               "gtyp_VGR".vertical_Axis.di_Target_Position := "gtyp_VGR".di_Pos_NFC_vertical - "gtyp_VGR".di_Offset_Pos_DSI_NFC_vertical;
               "gtyp_VGR".vertical_Axis.x_Start_Positioning := TRUE;
               //"gtyp_VGR".vertical_Axis.i_PWM := 800;

               IF ("gtyp_VGR".vertical_Axis.di_Actual_Position <= ("gtyp_VGR".di_Pos_NFC_vertical - "gtyp_VGR".di_Offset_Pos_DSI_NFC_vertical + "gtyp_VGR".vertical_Axis.Config.di_Pos_Window))
                   AND ("gtyp_VGR".vertical_Axis.di_Actual_Position >= ("gtyp_VGR".di_Pos_NFC_vertical - "gtyp_VGR".di_Offset_Pos_DSI_NFC_vertical - "gtyp_VGR".vertical_Axis.Config.di_Pos_Window))
                   AND "gtyp_VGR".vertical_Axis.x_Position_Reached THEN
                   "gtyp_VGR".vertical_Axis.x_Start_Positioning := FALSE;
                   #li_StepCase := 660;
               END_IF;

           660: // wait sequence
               #lx_Start_TON_Wait := TRUE;
               #lt_TON_Wait := T#500ms;

               IF #lfb_TON_Wait.Q THEN
                   #lx_Start_TON_Wait := FALSE;
                   #li_StepCase := 670;
               END_IF;

           670: // Position horizontal/rotate NFC

               "gtyp_VGR".horizontal_Axis.di_Target_Position := "gtyp_VGR".di_Pos_NFC_horizontal;
               "gtyp_VGR".horizontal_Axis.x_Start_Positioning := TRUE;
               "gtyp_VGR".rotate_Axis.di_Target_Position := "gtyp_VGR".di_Pos_NFC_rotate;
               "gtyp_VGR".rotate_Axis.x_Start_Positioning := TRUE;

               IF ("gtyp_VGR".horizontal_Axis.di_Actual_Position <= ("gtyp_VGR".di_Pos_NFC_horizontal + "gtyp_VGR".horizontal_Axis.Config.di_Pos_Window))
                   AND ("gtyp_VGR".horizontal_Axis.di_Actual_Position >= ("gtyp_VGR".di_Pos_NFC_horizontal - "gtyp_VGR".horizontal_Axis.Config.di_Pos_Window))
                   AND "gtyp_VGR".horizontal_Axis.x_Position_Reached THEN
                   "gtyp_VGR".horizontal_Axis.x_Start_Positioning := FALSE;
               END_IF;

               IF ("gtyp_VGR".rotate_Axis.di_Actual_Position <= ("gtyp_VGR".di_Pos_NFC_rotate + "gtyp_VGR".rotate_Axis.Config.di_Pos_Window))
                   AND ("gtyp_VGR".rotate_Axis.di_Actual_Position >= ("gtyp_VGR".di_Pos_NFC_rotate - "gtyp_VGR".rotate_Axis.Config.di_Pos_Window))
                   AND "gtyp_VGR".rotate_Axis.x_Position_Reached THEN
                   "gtyp_VGR".rotate_Axis.x_Start_Positioning := FALSE;
               END_IF;

               IF ("gtyp_VGR".horizontal_Axis.di_Actual_Position <= ("gtyp_VGR".di_Pos_NFC_horizontal + "gtyp_VGR".horizontal_Axis.Config.di_Pos_Window))
                   AND ("gtyp_VGR".horizontal_Axis.di_Actual_Position >= ("gtyp_VGR".di_Pos_NFC_horizontal - "gtyp_VGR".horizontal_Axis.Config.di_Pos_Window))
                   AND "gtyp_VGR".horizontal_Axis.x_Position_Reached
                   AND ("gtyp_VGR".rotate_Axis.di_Actual_Position <= ("gtyp_VGR".di_Pos_NFC_rotate + "gtyp_VGR".rotate_Axis.Config.di_Pos_Window))
                   AND ("gtyp_VGR".rotate_Axis.di_Actual_Position >= ("gtyp_VGR".di_Pos_NFC_rotate - "gtyp_VGR".rotate_Axis.Config.di_Pos_Window))
                   AND "gtyp_VGR".rotate_Axis.x_Position_Reached THEN
                   "gtyp_VGR".horizontal_Axis.x_Start_Positioning := FALSE;
                   "gtyp_VGR".rotate_Axis.x_Start_Positioning := FALSE;
                   #li_StepCase := 680;
               END_IF;

           680: // wait sequence
               #lx_Start_TON_Wait := TRUE;
               #lt_TON_Wait := T#500ms;

               IF #lfb_TON_Wait.Q THEN
                   #lx_Start_TON_Wait := FALSE;
                   #li_StepCase := 690;
               END_IF;

           690: // Position vertical NFC

               "gtyp_VGR".vertical_Axis.di_Target_Position := "gtyp_VGR".di_Pos_NFC_vertical;
               "gtyp_VGR".vertical_Axis.x_Start_Positioning := TRUE;
               //"gtyp_VGR".vertical_Axis.i_PWM := 500;

               IF ("gtyp_VGR".vertical_Axis.di_Actual_Position <= ("gtyp_VGR".di_Pos_NFC_vertical + "gtyp_VGR".vertical_Axis.Config.di_Pos_Window))
                   AND ("gtyp_VGR".vertical_Axis.di_Actual_Position >= ("gtyp_VGR".di_Pos_NFC_vertical - "gtyp_VGR".vertical_Axis.Config.di_Pos_Window))
                   AND "gtyp_VGR".vertical_Axis.x_Position_Reached THEN
                   "gtyp_VGR".vertical_Axis.x_Start_Positioning := FALSE;
                   //"gtyp_VGR".vertical_Axis.i_PWM := 800;
                   #li_StepCase := 700;
               END_IF;

           700: // Start delete/write/read NFC 
               "gtyp_VGR".x_NFC_Start_First := TRUE;

               IF "gtyp_VGR".x_NFC_Completed THEN
                   "gtyp_VGR".x_NFC_Start_First := FALSE;
                   #li_StepCase := 710;
               END_IF;

           710: // Position vertical pre NFC

               "gtyp_VGR".vertical_Axis.di_Target_Position := "gtyp_VGR".di_Pos_NFC_vertical - "gtyp_VGR".di_Offset_Pos_DSI_NFC_vertical;
               "gtyp_VGR".vertical_Axis.x_Start_Positioning := TRUE;
               //"gtyp_VGR".vertical_Axis.i_PWM := 800;

               IF ("gtyp_VGR".vertical_Axis.di_Actual_Position <= ("gtyp_VGR".di_Pos_NFC_vertical - "gtyp_VGR".di_Offset_Pos_DSI_NFC_vertical + "gtyp_VGR".vertical_Axis.Config.di_Pos_Window))
                   AND ("gtyp_VGR".vertical_Axis.di_Actual_Position >= ("gtyp_VGR".di_Pos_NFC_vertical - "gtyp_VGR".di_Offset_Pos_DSI_NFC_vertical - "gtyp_VGR".vertical_Axis.Config.di_Pos_Window))
                   AND "gtyp_VGR".vertical_Axis.x_Position_Reached THEN
                   "gtyp_VGR".vertical_Axis.x_Start_Positioning := FALSE;
                   #li_StepCase := 720;
               END_IF;

           720: // Position horizontal/rotate Color

               "gtyp_VGR".horizontal_Axis.di_Target_Position := "gtyp_VGR".di_Pos_Color_horizontal;
               "gtyp_VGR".horizontal_Axis.x_Start_Positioning := TRUE;
               "gtyp_VGR".rotate_Axis.di_Target_Position := "gtyp_VGR".di_Pos_Color_rotate;
               "gtyp_VGR".rotate_Axis.x_Start_Positioning := TRUE;

               IF ("gtyp_VGR".horizontal_Axis.di_Actual_Position <= ("gtyp_VGR".di_Pos_Color_horizontal + "gtyp_VGR".horizontal_Axis.Config.di_Pos_Window))
                   AND ("gtyp_VGR".horizontal_Axis.di_Actual_Position >= ("gtyp_VGR".di_Pos_Color_horizontal - "gtyp_VGR".horizontal_Axis.Config.di_Pos_Window))
                   AND "gtyp_VGR".horizontal_Axis.x_Position_Reached THEN
                   "gtyp_VGR".horizontal_Axis.x_Start_Positioning := FALSE;
               END_IF;

               IF ("gtyp_VGR".rotate_Axis.di_Actual_Position <= ("gtyp_VGR".di_Pos_Color_rotate + "gtyp_VGR".rotate_Axis.Config.di_Pos_Window))
                   AND ("gtyp_VGR".rotate_Axis.di_Actual_Position >= ("gtyp_VGR".di_Pos_Color_rotate - "gtyp_VGR".rotate_Axis.Config.di_Pos_Window))
                   AND "gtyp_VGR".rotate_Axis.x_Position_Reached THEN
                   "gtyp_VGR".rotate_Axis.x_Start_Positioning := FALSE;
               END_IF;

               IF ("gtyp_VGR".horizontal_Axis.di_Actual_Position <= ("gtyp_VGR".di_Pos_Color_horizontal + "gtyp_VGR".horizontal_Axis.Config.di_Pos_Window))
                   AND ("gtyp_VGR".horizontal_Axis.di_Actual_Position >= ("gtyp_VGR".di_Pos_Color_horizontal - "gtyp_VGR".horizontal_Axis.Config.di_Pos_Window))
                   AND "gtyp_VGR".horizontal_Axis.x_Position_Reached
                   AND ("gtyp_VGR".rotate_Axis.di_Actual_Position <= ("gtyp_VGR".di_Pos_Color_rotate + "gtyp_VGR".rotate_Axis.Config.di_Pos_Window))
                   AND ("gtyp_VGR".rotate_Axis.di_Actual_Position >= ("gtyp_VGR".di_Pos_Color_rotate - "gtyp_VGR".rotate_Axis.Config.di_Pos_Window))
                   AND "gtyp_VGR".rotate_Axis.x_Position_Reached THEN
                   "gtyp_VGR".horizontal_Axis.x_Start_Positioning := FALSE;
                   "gtyp_VGR".rotate_Axis.x_Start_Positioning := FALSE;
                   #li_StepCase := 730;
               END_IF;

           730: // wait sequence
               #lx_Start_TON_Wait := TRUE;
               #lt_TON_Wait := T#500ms;

               IF #lfb_TON_Wait.Q THEN
                   #lx_Start_TON_Wait := FALSE;
                   #li_StepCase := 740;
               END_IF;

           740: // Position vertical Color
               "gtyp_VGR".vertical_Axis.di_Target_Position := "gtyp_VGR".di_Pos_Color_vertical;
               "gtyp_VGR".vertical_Axis.x_Start_Positioning := TRUE;
               //"gtyp_VGR".vertical_Axis.i_PWM := 500;

               IF ("gtyp_VGR".vertical_Axis.di_Actual_Position <= ("gtyp_VGR".di_Pos_Color_vertical + "gtyp_VGR".vertical_Axis.Config.di_Pos_Window))
                   AND ("gtyp_VGR".vertical_Axis.di_Actual_Position >= ("gtyp_VGR".di_Pos_Color_vertical - "gtyp_VGR".vertical_Axis.Config.di_Pos_Window))
                   AND "gtyp_VGR".vertical_Axis.x_Position_Reached THEN
                   "gtyp_VGR".vertical_Axis.x_Start_Positioning := FALSE;
                   //"gtyp_VGR".vertical_Axis.i_PWM := 800;
                   #li_StepCase := 750;
               END_IF;

           750: // evaluate color workpiece
               #ls_Color := '';

               IF "IW_SSC_ColorSensor_A1" >= "gtyp_SSC".w_Threshold_Red_Blue THEN
                   //               IF "IW_SSC_ColorSensor" > 16000 AND "IW_SSC_ColorSensor" < 17500 THEN
                   #ls_Color := 'BLUE';
               ELSIF "IW_SSC_ColorSensor_A1" <= "gtyp_SSC".w_Threshold_White_Red THEN
                   //            ELSIF "IW_SSC_ColorSensor" > 5000 AND "IW_SSC_ColorSensor" < 11000 THEN
                   #ls_Color := 'WHITE';
               ELSIF "IW_SSC_ColorSensor_A1" > "gtyp_SSC".w_Threshold_White_Red AND "IW_SSC_ColorSensor_A1" < "gtyp_SSC".w_Threshold_Red_Blue THEN
                   //            ELSIF "IW_SSC_ColorSensor" > 11000 AND "IW_SSC_ColorSensor" < 16000 THEN
                   #ls_Color := 'RED';
               END_IF;

               #li_Return_LDT := RD_SYS_T(#ldt_MQTT);
               "gtyp_VGR".History[2].ldt_ts := DT_TO_LDT(#ldt_MQTT);
               "gtyp_VGR".History[2].i_code := 200;
               "gtyp_VGR".Workpiece.s_type := #ls_Color;

               #lx_Start_TON_Wait := TRUE;
               #lt_TON_Wait := T#500ms;

               IF #lfb_TON_Wait.Q THEN
                   #lx_Start_TON_Wait := FALSE;
                   #li_StepCase := 760;
               END_IF;

           760: // Position vertical pre NFC
               "gtyp_VGR".vertical_Axis.di_Target_Position := "gtyp_VGR".di_Pos_NFC_vertical - "gtyp_VGR".di_Offset_Pos_DSI_NFC_vertical;
               "gtyp_VGR".vertical_Axis.x_Start_Positioning := TRUE;
               //"gtyp_VGR".vertical_Axis.i_PWM := 500;

               IF ("gtyp_VGR".vertical_Axis.di_Actual_Position <= ("gtyp_VGR".di_Pos_NFC_vertical - "gtyp_VGR".di_Offset_Pos_DSI_NFC_vertical + "gtyp_VGR".vertical_Axis.Config.di_Pos_Window))
                   AND ("gtyp_VGR".vertical_Axis.di_Actual_Position >= ("gtyp_VGR".di_Pos_NFC_vertical - "gtyp_VGR".di_Offset_Pos_DSI_NFC_vertical - "gtyp_VGR".vertical_Axis.Config.di_Pos_Window))
                   AND "gtyp_VGR".vertical_Axis.x_Position_Reached THEN
                   "gtyp_VGR".vertical_Axis.x_Start_Positioning := FALSE;
                   //"gtyp_VGR".vertical_Axis.i_PWM := 800;
                   #li_StepCase := 770;
               END_IF;

           770: // wait sequence
               #lx_Start_TON_Wait := TRUE;
               #lt_TON_Wait := T#500ms;

               IF #lfb_TON_Wait.Q THEN
                   #lx_Start_TON_Wait := FALSE;
                   #li_StepCase := 780;
               END_IF;

           780: // Position horizontal/rotate NFC

               "gtyp_VGR".horizontal_Axis.di_Target_Position := "gtyp_VGR".di_Pos_NFC_horizontal;
               "gtyp_VGR".horizontal_Axis.x_Start_Positioning := TRUE;
               "gtyp_VGR".rotate_Axis.di_Target_Position := "gtyp_VGR".di_Pos_NFC_rotate;
               "gtyp_VGR".rotate_Axis.x_Start_Positioning := TRUE;

               IF ("gtyp_VGR".horizontal_Axis.di_Actual_Position <= ("gtyp_VGR".di_Pos_NFC_horizontal + "gtyp_VGR".horizontal_Axis.Config.di_Pos_Window))
                   AND ("gtyp_VGR".horizontal_Axis.di_Actual_Position >= ("gtyp_VGR".di_Pos_NFC_horizontal - "gtyp_VGR".horizontal_Axis.Config.di_Pos_Window))
                   AND "gtyp_VGR".horizontal_Axis.x_Position_Reached THEN
                   "gtyp_VGR".horizontal_Axis.x_Start_Positioning := FALSE;
               END_IF;

               IF ("gtyp_VGR".rotate_Axis.di_Actual_Position <= ("gtyp_VGR".di_Pos_NFC_rotate + "gtyp_VGR".rotate_Axis.Config.di_Pos_Window))
                   AND ("gtyp_VGR".rotate_Axis.di_Actual_Position >= ("gtyp_VGR".di_Pos_NFC_rotate - "gtyp_VGR".rotate_Axis.Config.di_Pos_Window))
                   AND "gtyp_VGR".rotate_Axis.x_Position_Reached THEN
                   "gtyp_VGR".rotate_Axis.x_Start_Positioning := FALSE;
               END_IF;

               IF ("gtyp_VGR".horizontal_Axis.di_Actual_Position <= ("gtyp_VGR".di_Pos_NFC_horizontal + "gtyp_VGR".horizontal_Axis.Config.di_Pos_Window))
                   AND ("gtyp_VGR".horizontal_Axis.di_Actual_Position >= ("gtyp_VGR".di_Pos_NFC_horizontal - "gtyp_VGR".horizontal_Axis.Config.di_Pos_Window))
                   AND "gtyp_VGR".horizontal_Axis.x_Position_Reached
                   AND ("gtyp_VGR".rotate_Axis.di_Actual_Position <= ("gtyp_VGR".di_Pos_NFC_rotate + "gtyp_VGR".rotate_Axis.Config.di_Pos_Window))
                   AND ("gtyp_VGR".rotate_Axis.di_Actual_Position >= ("gtyp_VGR".di_Pos_NFC_rotate - "gtyp_VGR".rotate_Axis.Config.di_Pos_Window))
                   AND "gtyp_VGR".rotate_Axis.x_Position_Reached THEN
                   "gtyp_VGR".horizontal_Axis.x_Start_Positioning := FALSE;
                   "gtyp_VGR".vertical_Axis.x_Start_Positioning := FALSE;
                   "gtyp_VGR".rotate_Axis.x_Start_Positioning := FALSE;
                   #li_StepCase := 790;
               END_IF;

           790: // wait sequence
               #lx_Start_TON_Wait := TRUE;
               #lt_TON_Wait := T#500ms;

               IF #lfb_TON_Wait.Q THEN
                   #lx_Start_TON_Wait := FALSE;
                   #li_StepCase := 800;
               END_IF;

           800: // Position vertical NFC

               "gtyp_VGR".vertical_Axis.di_Target_Position := "gtyp_VGR".di_Pos_NFC_vertical;
               "gtyp_VGR".vertical_Axis.x_Start_Positioning := TRUE;
               //"gtyp_VGR".vertical_Axis.i_PWM := 500;

               IF ("gtyp_VGR".vertical_Axis.di_Actual_Position <= ("gtyp_VGR".di_Pos_NFC_vertical + "gtyp_VGR".vertical_Axis.Config.di_Pos_Window))
                   AND ("gtyp_VGR".vertical_Axis.di_Actual_Position >= ("gtyp_VGR".di_Pos_NFC_vertical - "gtyp_VGR".vertical_Axis.Config.di_Pos_Window))
                   AND "gtyp_VGR".vertical_Axis.x_Position_Reached THEN
                   "gtyp_VGR".vertical_Axis.x_Start_Positioning := FALSE;
                   //"gtyp_VGR".vertical_Axis.i_PWM := 800;
                   #li_StepCase := 810;
               END_IF;

           810: // Start write/read NFC Color

               "gtyp_VGR".x_NFC_Start := TRUE;

               IF "gtyp_VGR".x_NFC_Completed THEN
                   "gtyp_VGR".x_NFC_Start := FALSE;
                   #li_StepCase := 820;
               END_IF;

           820: // Position vertical pre NFC

               "gtyp_VGR".vertical_Axis.di_Target_Position := "gtyp_VGR".di_Pos_NFC_vertical - "gtyp_VGR".di_Offset_Pos_DSI_NFC_vertical;
               "gtyp_VGR".vertical_Axis.x_Start_Positioning := TRUE;
               //"gtyp_VGR".vertical_Axis.i_PWM := 500;

               IF ("gtyp_VGR".vertical_Axis.di_Actual_Position <= ("gtyp_VGR".di_Pos_NFC_vertical - "gtyp_VGR".di_Offset_Pos_DSI_NFC_vertical + "gtyp_VGR".vertical_Axis.Config.di_Pos_Window))
                   AND ("gtyp_VGR".vertical_Axis.di_Actual_Position >= ("gtyp_VGR".di_Pos_NFC_vertical - "gtyp_VGR".di_Offset_Pos_DSI_NFC_vertical - "gtyp_VGR".vertical_Axis.Config.di_Pos_Window))
                   AND "gtyp_VGR".vertical_Axis.x_Position_Reached THEN
                   "gtyp_VGR".vertical_Axis.x_Start_Positioning := FALSE;
                   //"gtyp_VGR".vertical_Axis.i_PWM := 800;
                   #li_StepCase := 830;
               END_IF;

           830: // wait sequence
               #lx_Start_TON_Wait := TRUE;
               #lt_TON_Wait := T#500ms;

               IF #lfb_TON_Wait.Q THEN
                   #lx_Start_TON_Wait := FALSE;
                   #li_StepCase := 840;
               END_IF;

           840: // Position rotate HBW and homing horizontal/vertical axis
               "gtyp_VGR".rotate_Axis.di_Target_Position := "gtyp_VGR".di_Pos_HBW_rotate;
               "gtyp_VGR".rotate_Axis.x_Start_Positioning := TRUE;

               "gtyp_VGR".horizontal_Axis.x_Reference := TRUE;
               "gtyp_VGR".vertical_Axis.x_Reference := TRUE;

               IF ("gtyp_VGR".rotate_Axis.di_Actual_Position <= ("gtyp_VGR".di_Pos_HBW_rotate + "gtyp_VGR".rotate_Axis.Config.di_Pos_Window))
                   AND ("gtyp_VGR".rotate_Axis.di_Actual_Position >= ("gtyp_VGR".di_Pos_HBW_rotate - "gtyp_VGR".rotate_Axis.Config.di_Pos_Window))
                   AND "gtyp_VGR".rotate_Axis.x_Position_Reached THEN
                   "gtyp_VGR".rotate_Axis.x_Start_Positioning := FALSE;
               END_IF;

               IF NOT "gtyp_VGR".horizontal_Axis.x_Referenced AND NOT "gtyp_VGR".vertical_Axis.x_Referenced THEN
                   #li_StepCase := 850;
               END_IF;

           850: // Position rotate HBW reached and homed horizontal/vertical axis

               IF ("gtyp_VGR".rotate_Axis.di_Actual_Position <= ("gtyp_VGR".di_Pos_HBW_rotate + "gtyp_VGR".rotate_Axis.Config.di_Pos_Window))
                   AND ("gtyp_VGR".rotate_Axis.di_Actual_Position >= ("gtyp_VGR".di_Pos_HBW_rotate - "gtyp_VGR".rotate_Axis.Config.di_Pos_Window))
                   AND "gtyp_VGR".rotate_Axis.x_Position_Reached THEN
                   "gtyp_VGR".rotate_Axis.x_Start_Positioning := FALSE;
               END_IF;

               IF "gtyp_VGR".horizontal_Axis.x_Referenced THEN
                   "gtyp_VGR".horizontal_Axis.x_Reference := FALSE;
               END_IF;
               IF "gtyp_VGR".vertical_Axis.x_Referenced THEN
                   "gtyp_VGR".vertical_Axis.x_Reference := FALSE;
               END_IF;
               IF "gtyp_VGR".horizontal_Axis.x_Referenced
                   AND "gtyp_VGR".vertical_Axis.x_Referenced
                   AND ("gtyp_VGR".rotate_Axis.di_Actual_Position <= ("gtyp_VGR".di_Pos_HBW_rotate + "gtyp_VGR".rotate_Axis.Config.di_Pos_Window))
                   AND ("gtyp_VGR".rotate_Axis.di_Actual_Position >= ("gtyp_VGR".di_Pos_HBW_rotate - "gtyp_VGR".rotate_Axis.Config.di_Pos_Window))
                   AND "gtyp_VGR".rotate_Axis.x_Position_Reached THEN
                   "gtyp_VGR".horizontal_Axis.x_Reference := FALSE;
                   "gtyp_VGR".vertical_Axis.x_Reference := FALSE;
                   "gtyp_VGR".rotate_Axis.x_Start_Positioning := FALSE;
                   #li_StepCase := 860;
               END_IF;

           860: // wait sequence
               #lx_Start_TON_Wait := TRUE;
               #lt_TON_Wait := T#500ms;

               IF #lfb_TON_Wait.Q THEN
                   #lx_Start_TON_Wait := FALSE;
                   #li_StepCase := 870;
               END_IF;

           870: // Position horizontal HBW

               "gtyp_VGR".horizontal_Axis.di_Target_Position := "gtyp_VGR".di_Pos_HBW_horizontal;
               "gtyp_VGR".horizontal_Axis.x_Start_Positioning := TRUE;

               IF ("gtyp_VGR".horizontal_Axis.di_Actual_Position <= ("gtyp_VGR".di_Pos_HBW_horizontal + "gtyp_VGR".horizontal_Axis.Config.di_Pos_Window))
                   AND ("gtyp_VGR".horizontal_Axis.di_Actual_Position >= ("gtyp_VGR".di_Pos_HBW_horizontal - "gtyp_VGR".horizontal_Axis.Config.di_Pos_Window))
                   AND "gtyp_VGR".horizontal_Axis.x_Position_Reached THEN
                   "gtyp_VGR".horizontal_Axis.x_Start_Positioning := FALSE;
                   #li_StepCase := 880;
               END_IF;

           880: // container available start drop down
               IF "gtyp_HBW".x_HBW_Container_Available THEN
                   #li_StepCase := 890;
               END_IF;

           890: // Position vertical discard HBW
               "gtyp_VGR".vertical_Axis.di_Target_Position := "gtyp_VGR".di_Pos_HBW_Discard_vertical;
               "gtyp_VGR".vertical_Axis.x_Start_Positioning := TRUE;
               //"gtyp_VGR".vertical_Axis.i_PWM := 500;

               IF ("gtyp_VGR".vertical_Axis.di_Actual_Position <= ("gtyp_VGR".di_Pos_HBW_Discard_vertical + "gtyp_VGR".vertical_Axis.Config.di_Pos_Window))
                   AND ("gtyp_VGR".vertical_Axis.di_Actual_Position >= ("gtyp_VGR".di_Pos_HBW_Discard_vertical - "gtyp_VGR".vertical_Axis.Config.di_Pos_Window))
                   AND "gtyp_VGR".vertical_Axis.x_Position_Reached THEN
                   "gtyp_VGR".vertical_Axis.x_Start_Positioning := FALSE;
                   //"gtyp_VGR".vertical_Axis.i_PWM := 800;
                   #li_StepCase := 900;
               END_IF;

           900: // turn off vacuum
               "QX_VGR_ValveVacuum_Q8" := FALSE;
               #li_StepCase := 910;

           910: // turn off compressor
               "QX_VGR_Compressor_Q7" := FALSE;
               "gtyp_VGR".x_HBW_Discards := TRUE;

               #lx_Start_TON_Wait := TRUE;
               #lt_TON_Wait := T#500ms;

               IF #lfb_TON_Wait.Q AND "gtyp_HBW".x_HBW_Discards_Accepted THEN
                   #lx_State_activ := FALSE;
                   #ls_Target := '';
                   "gtyp_VGR".x_HBW_Discards := FALSE;
                   "gtyp_VGR".x_HBW_Storage := FALSE;
                   #lx_Start_TON_Wait := FALSE;
                   #li_StepCase := 920;
               END_IF;

           920: // homing vertical axis
               "gtyp_VGR".vertical_Axis.x_Reference := TRUE;

               IF NOT "gtyp_VGR".vertical_Axis.x_Referenced THEN
                   #li_StepCase := 930;
               END_IF;

           930: // homed vertical axis
               IF "gtyp_VGR".vertical_Axis.x_Referenced THEN
                   "gtyp_VGR".vertical_Axis.x_Reference := FALSE;
                   #li_StepCase := 940;
               END_IF;

           940: // homing horizontal axis
               "gtyp_VGR".horizontal_Axis.x_Reference := TRUE;

               IF NOT "gtyp_VGR".horizontal_Axis.x_Referenced THEN
                   #li_StepCase := 950;
               END_IF;

           950: // homed horizontal axis
               IF "gtyp_VGR".horizontal_Axis.x_Referenced THEN
                   "gtyp_VGR".horizontal_Axis.x_Reference := FALSE;
                   #li_StepCase := 960;
               END_IF;

           960: // wait sequence
               #lx_Start_TON_Wait := TRUE;
               #lt_TON_Wait := T#500ms;

               IF #lfb_TON_Wait.Q AND "gtyp_HBW".x_HBW_Discards_Accepted THEN
                   "gtyp_VGR".x_HBW_Discards := FALSE;
                   #lx_Start_TON_Wait := FALSE;
                   "gtyp_VGR".Workpiece.s_id := '';
                   "gtyp_VGR".Workpiece.s_state := '';
                   "gtyp_VGR".Workpiece.s_type := '';
                   FOR #ti_Counter := 1 TO 8 DO
                       // Statement section FOR
                       "gtyp_VGR".History[#ti_Counter].i_code := 0;
                       "gtyp_VGR".History[#ti_Counter].ldt_ts := DT#1990-01-01-00:00:00;
                   END_FOR;
                   #li_StepCase := 0;
               END_IF;

           1200:// homing vertical axis
               "gtyp_VGR".Workpiece.s_id := '0';
               "gtyp_VGR".Workpiece.s_state := '';
               "gtyp_VGR".Workpiece.s_type := '';
               FOR #ti_Counter := 1 TO 8 DO
                   "gtyp_VGR".History[#ti_Counter].i_code := 0;
                   "gtyp_VGR".History[#ti_Counter].ldt_ts := DT#1990-01-01-00:00:00;
               END_FOR;

               IF "gtyp_HBW".x_HBW_Container_Available THEN
                   "gtyp_VGR".x_HBW_Discards := TRUE;
               END_IF;

               IF "gtyp_HBW".x_HBW_Discards_Accepted OR "gtyp_HBW".x_HBW_PickedUp_Accepted THEN
                   "gtyp_VGR".x_HBW_Discards := FALSE;
                   "gtyp_VGR".x_HBW_PickedUp := FALSE;
                   "gtyp_HBW".x_HBW_Discards_Accepted := FALSE;
                   "gtyp_HBW".x_HBW_PickedUp_Accepted := FALSE;
               END_IF;

               #li_Lights := 2;
               "gtyp_VGR".vertical_Axis.x_Reference := TRUE;

               IF NOT "gtyp_VGR".vertical_Axis.x_Referenced THEN
                   #li_StepCase := 1210;
               END_IF;

           1210: // homed vertical axis
               IF "gtyp_VGR".vertical_Axis.x_Referenced THEN
                   "gtyp_VGR".vertical_Axis.x_Reference := FALSE;
                   #li_StepCase := 1220;
               END_IF;

           1220: // homing horizontal axis
               "gtyp_VGR".horizontal_Axis.x_Reference := TRUE;

               IF NOT "gtyp_VGR".horizontal_Axis.x_Referenced THEN
                   #li_StepCase := 1230;
               END_IF;

           1230: // homed horizontal axis
               IF "gtyp_VGR".horizontal_Axis.x_Referenced THEN
                   "gtyp_VGR".horizontal_Axis.x_Reference := FALSE;
                   #li_StepCase := 1240;
               END_IF;

           1240: // homing rotate axis
               "gtyp_VGR".rotate_Axis.x_Reference := TRUE;

               IF NOT "gtyp_VGR".rotate_Axis.x_Referenced THEN
                   #li_StepCase := 1250;
               END_IF;

           1250: // homed horizontal axis
               IF "gtyp_VGR".rotate_Axis.x_Referenced THEN
                   "gtyp_VGR".rotate_Axis.x_Reference := FALSE;
                   #li_StepCase := 1260;
               END_IF;

           1260: // Position vertical/horizontal/rotate NiO
               "gtyp_VGR".horizontal_Axis.di_Target_Position := "gtyp_VGR".di_Pos_NiO_horizontal;
               "gtyp_VGR".horizontal_Axis.x_Start_Positioning := TRUE;
               "gtyp_VGR".vertical_Axis.di_Target_Position := "gtyp_VGR".di_Pos_NiO_vertical;
               "gtyp_VGR".vertical_Axis.x_Start_Positioning := TRUE;
               //"gtyp_VGR".vertical_Axis.i_PWM := 500;
               "gtyp_VGR".rotate_Axis.di_Target_Position := "gtyp_VGR".di_Pos_NiO_rotate;
               "gtyp_VGR".rotate_Axis.x_Start_Positioning := TRUE;

               IF ("gtyp_VGR".horizontal_Axis.di_Actual_Position <= ("gtyp_VGR".di_Pos_NiO_horizontal + "gtyp_VGR".horizontal_Axis.Config.di_Pos_Window))
                   AND ("gtyp_VGR".horizontal_Axis.di_Actual_Position >= ("gtyp_VGR".di_Pos_NiO_horizontal - "gtyp_VGR".horizontal_Axis.Config.di_Pos_Window))
                   AND "gtyp_VGR".horizontal_Axis.x_Position_Reached THEN
                   "gtyp_VGR".horizontal_Axis.x_Start_Positioning := FALSE;
               END_IF;

               IF ("gtyp_VGR".vertical_Axis.di_Actual_Position <= ("gtyp_VGR".di_Pos_NiO_vertical + "gtyp_VGR".vertical_Axis.Config.di_Pos_Window))
                   AND ("gtyp_VGR".vertical_Axis.di_Actual_Position >= ("gtyp_VGR".di_Pos_NiO_vertical - "gtyp_VGR".vertical_Axis.Config.di_Pos_Window))
                   AND "gtyp_VGR".vertical_Axis.x_Position_Reached THEN
                   "gtyp_VGR".vertical_Axis.x_Start_Positioning := FALSE;
               END_IF;

               IF ("gtyp_VGR".rotate_Axis.di_Actual_Position <= ("gtyp_VGR".di_Pos_NiO_rotate + "gtyp_VGR".rotate_Axis.Config.di_Pos_Window))
                   AND ("gtyp_VGR".rotate_Axis.di_Actual_Position >= ("gtyp_VGR".di_Pos_NiO_rotate - "gtyp_VGR".rotate_Axis.Config.di_Pos_Window))
                   AND "gtyp_VGR".rotate_Axis.x_Position_Reached THEN
                   "gtyp_VGR".rotate_Axis.x_Start_Positioning := FALSE;
               END_IF;

               IF ("gtyp_VGR".horizontal_Axis.di_Actual_Position <= ("gtyp_VGR".di_Pos_NiO_horizontal + "gtyp_VGR".horizontal_Axis.Config.di_Pos_Window))
                   AND ("gtyp_VGR".horizontal_Axis.di_Actual_Position >= ("gtyp_VGR".di_Pos_NiO_horizontal - "gtyp_VGR".horizontal_Axis.Config.di_Pos_Window))
                   AND "gtyp_VGR".horizontal_Axis.x_Position_Reached
                   AND ("gtyp_VGR".vertical_Axis.di_Actual_Position <= ("gtyp_VGR".di_Pos_NiO_vertical + "gtyp_VGR".vertical_Axis.Config.di_Pos_Window))
                   AND ("gtyp_VGR".vertical_Axis.di_Actual_Position >= ("gtyp_VGR".di_Pos_NiO_vertical - "gtyp_VGR".vertical_Axis.Config.di_Pos_Window))
                   AND "gtyp_VGR".vertical_Axis.x_Position_Reached
                   AND ("gtyp_VGR".rotate_Axis.di_Actual_Position <= ("gtyp_VGR".di_Pos_NiO_rotate + "gtyp_VGR".rotate_Axis.Config.di_Pos_Window))
                   AND ("gtyp_VGR".rotate_Axis.di_Actual_Position >= ("gtyp_VGR".di_Pos_NiO_rotate - "gtyp_VGR".rotate_Axis.Config.di_Pos_Window))
                   AND "gtyp_VGR".rotate_Axis.x_Position_Reached THEN
                   "gtyp_VGR".horizontal_Axis.x_Start_Positioning := FALSE;
                   "gtyp_VGR".vertical_Axis.x_Start_Positioning := FALSE;
                   "gtyp_VGR".rotate_Axis.x_Start_Positioning := FALSE;
                   //"gtyp_VGR".vertical_Axis.i_PWM := 800;
                   #li_StepCase := 1270;
               END_IF;

           1270: // turn off vacuum
               "QX_VGR_ValveVacuum_Q8" := FALSE;
               #li_StepCase := 1280;

           1280: // turn off compressor

               #lx_Start_TON_Wait := TRUE;
               #lt_TON_Wait := T#1000ms;

               IF #lfb_TON_Wait.Q THEN
                   "QX_VGR_Compressor_Q7" := FALSE;
                   #lx_Start_TON_Wait := FALSE;
                   "gtyp_VGR".x_Workpiece_NiO := FALSE;
                   "gtyp_VGR".x_HBW_Discards := FALSE;
                   #li_Lights := 1;
                   #li_StepCase := 0;
               END_IF;
               // Statement section ELSE       
           ELSE
               ;
       END_CASE;

   ELSE
       "gtyp_VGR".Workpiece.s_id := '';
       "gtyp_VGR".Workpiece.s_state := '';
       "gtyp_VGR".Workpiece.s_type := '';
       // Order State
       "gtyp_VGR".x_State_Process := FALSE;
       "gtyp_Interface_Dashboard".Subscribe.State_Order.ldt_ts := DT_TO_LDT(#ldt_MQTT);
       "gtyp_Interface_Dashboard".Subscribe.State_Order.s_state := 'WAITING_FOR_ORDER';
       "gtyp_Interface_Dashboard".Subscribe.State_Order.s_type := '';
       FOR #ti_Counter := 1 TO 8 DO
           "gtyp_VGR".History[#ti_Counter].i_code := 0;
           "gtyp_VGR".History[#ti_Counter].ldt_ts := DT#1990-01-01-00:00:00;
       END_FOR;

       "gtyp_VGR".x_Start_Park_Position := FALSE;
       "gtyp_VGR".x_Park_Position_Reached := FALSE;
       "gtyp_VGR".x_NFC_Start_First := FALSE;
       "gtyp_VGR".x_NFC_Start := FALSE;
       "gtyp_VGR".x_NFC_Completed := FALSE;
       "gtyp_VGR".x_HBW_Storage := FALSE;
       "gtyp_VGR".x_HBW_Outsource := FALSE;
       "gtyp_VGR".s_HBW_Outsource_Typ := '';
       "gtyp_VGR".x_HBW_Discards := FALSE;
       "gtyp_VGR".x_HBW_PickedUp := FALSE;
       "gtyp_VGR".x_MPO_Req_Discard := FALSE;
       "gtyp_VGR".x_MPO_Discards := FALSE;
       "gtyp_VGR".x_Ready_For_Outsource := FALSE;
       "gtyp_VGR".x_State_Process := FALSE;
       "gtyp_VGR".x_Workpiece_NiO := FALSE;

       "gtyp_VGR".x_Ready_For_Order := TRUE;

       #li_Lights := 1;
       #lx_Init := TRUE;
   END_IF;
END_FUNCTION_BLOCK

FUNCTION_BLOCK "PRG_NFC"   // FB8, SCL
TITLE = Program NFC
{ S7_Optimized_Access := 'TRUE' }
AUTHOR : A.Schaefer
VERSION : 0.0
   VAR
      lx_Init : Bool;
      lx_Start : Bool;
      lx_Time_Wait : Bool;
      lx_Time_Error : Bool;
      li_StepCase : Int;
      ldt_MQTT : Date_And_Time;
      ldt_Delete_old : LDT;
      ldt_Read_old : LDT;
      li_Return_LDT : Int;
      lfb_TON_Error : TON_TIME;
      lfb_TON_Wait : TON_TIME;
   END_VAR
BEGIN
   IF #lx_Init THEN

       // runtime monitoring error
       #lfb_TON_Error(IN := #lx_Time_Error,
                      PT := T#30s);

       // runtime monitoring read uid
       #lfb_TON_Wait(IN := #lx_Time_Wait,
                     PT := T#5s);

       // step chain NFC
       CASE #li_StepCase OF

           0:  // init
               #lx_Time_Wait := FALSE;
               "gtyp_VGR"."x_NFC_Completed" := FALSE;

               // delete and write first state to chip
               IF "gtyp_VGR".x_NFC_Start_First AND NOT "gtyp_VGR".x_Workpiece_NiO THEN
                   "gtyp_Interface_TXT_Controler".Subscribe.State_NFC_Device.Workpiece.s_state := '';
                   "gtyp_Interface_TXT_Controler".Subscribe.State_NFC_Device.Workpiece.s_type := '';

                   "gtyp_Interface_TXT_Controler".Publish.ActionButtonNFCModule.s_cmd := '';
                   #li_StepCase := 10;
                   // write color or processed finished to chip
               ELSIF "gtyp_VGR".x_NFC_Start AND NOT "gtyp_VGR".x_Workpiece_NiO THEN
                   "gtyp_Interface_TXT_Controler".Publish.ActionButtonNFCModule.s_cmd := '';
                   #li_StepCase := 40;
                   // read chip for delete HBW
               ELSIF "QX_SSC_LED_Green_Q5" AND NOT "gtyp_VGR".x_Workpiece_NiO THEN
                   #ldt_Read_old := "gtyp_Interface_Dashboard".Publish.ActionButtonNFCModule.ldt_ts;
                   "gtyp_VGR".x_NFC_Start_First := FALSE;
                   "gtyp_VGR".x_NFC_Start := FALSE;
                   "gtyp_Interface_TXT_Controler".Publish.ActionButtonNFCModule.s_cmd := '';
                   #li_StepCase := 60;
               END_IF;

           10: // delete

               "gtyp_Interface_TXT_Controler".Publish.ActionButtonNFCModule.s_cmd := 'delete';
               #li_Return_LDT := RD_SYS_T(#ldt_MQTT);
               "gtyp_Interface_TXT_Controler".Publish.ActionButtonNFCModule.ldt_ts := DT_TO_LDT(#ldt_MQTT);

               #li_StepCase := 20;

           20: // wait to answer from dashboard
               #lx_Time_Error := TRUE;
               IF ("gtyp_Interface_TXT_Controler".Subscribe.State_NFC_Device.ldt_ts > "gtyp_Interface_TXT_Controler".Publish.ActionButtonNFCModule.ldt_ts)
                   AND ("gtyp_Interface_TXT_Controler".Subscribe.State_NFC_Device.Workpiece.s_type = 'NONE')
                   AND ("gtyp_Interface_TXT_Controler".Subscribe.State_NFC_Device.Workpiece.s_state <> '')
                   AND ("gtyp_Interface_TXT_Controler".Subscribe.State_NFC_Device.Workpiece.s_id <> '') THEN
                   "gtyp_VGR".Workpiece.s_id := "gtyp_Interface_TXT_Controler".Subscribe.State_NFC_Device.Workpiece.s_id;
                   #lx_Time_Error := FALSE;
                   #li_StepCase := 30;
               END_IF;
               // runtime error
               IF #lfb_TON_Error.Q THEN
                   #lx_Time_Error := FALSE;
                   "gtyp_VGR".x_Workpiece_NiO := TRUE;
                   #li_StepCase := 0;
               END_IF;


           30: // wait of answer 
               IF "gtyp_Interface_TXT_Controler".Subscribe.State_NFC_Device.Workpiece.s_id <> '' THEN
                   #li_StepCase := 40;
               END_IF;

           40:  // write
               "gtyp_Interface_TXT_Controler".Publish.ActionButtonNFCModule.History := "gtyp_VGR".History;
               "gtyp_Interface_TXT_Controler".Publish.ActionButtonNFCModule.Workpiece.s_type := "gtyp_VGR".Workpiece.s_type;
               "gtyp_Interface_TXT_Controler".Publish.ActionButtonNFCModule.Workpiece.s_state := "gtyp_VGR".Workpiece.s_state;

               #li_Return_LDT := RD_SYS_T(#ldt_MQTT);

               "gtyp_Interface_TXT_Controler".Publish.ActionButtonNFCModule.s_cmd := 'write';
               "gtyp_Interface_TXT_Controler".Publish.ActionButtonNFCModule.ldt_ts := DT_TO_LDT(#ldt_MQTT);

               #li_StepCase := 50;

           50: // wait of answer write 
               #lx_Time_Error := TRUE;
               IF ("gtyp_Interface_TXT_Controler".Subscribe.State_NFC_Device.ldt_ts > "gtyp_Interface_TXT_Controler".Publish.ActionButtonNFCModule.ldt_ts) THEN
                   #lx_Time_Error := FALSE;
                   #li_StepCase := 80;
               END_IF;
               // runtime error
               IF #lfb_TON_Error.Q THEN
                   #lx_Time_Error := FALSE;
                   "gtyp_VGR".x_Workpiece_NiO := TRUE;
                   #li_StepCase := 0;
               END_IF;

           60: // read uid cmd

               #li_Return_LDT := RD_SYS_T(#ldt_MQTT);

               "gtyp_Interface_TXT_Controler".Publish.ActionButtonNFCModule.s_cmd := 'read_uid';
               "gtyp_Interface_TXT_Controler".Publish.ActionButtonNFCModule.ldt_ts := DT_TO_LDT(#ldt_MQTT);
               #lx_Time_Wait := TRUE;
               #li_StepCase := 70;

           70: // wait of answer read_uid 
               IF NOT "QX_SSC_LED_Green_Q5" OR #lfb_TON_Wait.Q OR ("gtyp_Interface_TXT_Controler".Subscribe.State_NFC_Device.ldt_ts > "gtyp_Interface_TXT_Controler".Publish.ActionButtonNFCModule.ldt_ts) THEN
                   IF LEN("gtyp_Interface_TXT_Controler".Subscribe.State_NFC_Device.Workpiece.s_id) = 8 THEN
                       "gtyp_Setup".x_Clean_Rack_HBW := TRUE;
                   END_IF;
                   #lx_Time_Wait := FALSE;
                   "gtyp_Interface_TXT_Controler".Subscribe.State_NFC_Device.Workpiece.s_id := '';
                   #li_StepCase := 0;
               END_IF;

           80: // completed

               "gtyp_VGR"."x_NFC_Completed" := TRUE;

               IF NOT "gtyp_VGR".x_NFC_Start AND NOT "gtyp_VGR".x_NFC_Start_First THEN
                   "gtyp_VGR"."x_NFC_Completed" := FALSE;
                   #lx_Start := FALSE;
                   #li_StepCase := 0;
               END_IF;

               // Statement section ELSE
           ELSE
               ;
       END_CASE;

   ELSE
       #lx_Init := TRUE;
   END_IF;
END_FUNCTION_BLOCK

FUNCTION_BLOCK "FB_INC_DEC"   // FB9, SCL
TITLE = Funktionblock Increment decodition
{ S7_Optimized_Access := 'TRUE' }
AUTHOR : A.Schaefer
VERSION : 0.0
   VAR_INPUT
      inx_CHa : Bool := FALSE;
      inx_CHb : Bool := FALSE;
      inx_RST : Bool := FALSE;
      ini_Ref_Wert : Int := 0;
   END_VAR
   VAR_OUTPUT
      outx_dir : Bool := FALSE;
      outi_cnt : Int := 0;
   END_VAR
   VAR
      lx_edgea : Bool := FALSE;
      lx_clka : Bool;
      lx_clkb : Bool;
      lx_edgeb : Bool;
      lx_axb : Bool;
      lx_dir : Bool;
      li_cnt : Int;
   END_VAR
BEGIN

   #lx_axb := #inx_CHa XOR #inx_CHb;

   (* create pulses for channel a *)
   #lx_clka := #inx_CHa XOR #lx_edgea;
   #lx_edgea := #inx_CHa;

   #lx_clkb := #inx_CHb XOR #lx_edgeb;
   #lx_edgeb := #inx_CHb;

   (* create pulses for both channels *)
   #lx_clka := #lx_clka OR #lx_clkb;

   (* set the direction output *)
   IF #lx_axb AND #lx_clka THEN
       #lx_dir := TRUE;
   END_IF;
   IF #lx_axb AND #lx_clkb THEN
       #lx_dir := FALSE;
   END_IF;

   (* increment or decrement the counter *)
   IF #lx_clka AND #lx_dir THEN
       #li_cnt := #li_cnt + 1;
   END_IF;
   IF #lx_clka AND NOT #lx_dir THEN
       #li_cnt := #li_cnt - 1;
   END_IF;

   (* reset the counter if rst active *)
   IF #inx_RST THEN
       #li_cnt := #ini_Ref_Wert;
   END_IF;

   #outx_dir := #lx_dir;
   #outi_cnt := #li_cnt;
END_FUNCTION_BLOCK

FUNCTION_BLOCK "PRG_VGR_Set_Positioning"   // FB10, SCL
TITLE = Program Set Positioning VGR
{ S7_Optimized_Access := 'TRUE' }
AUTHOR : A.Schaefer
VERSION : 0.0
   VAR
      lx_Init : Bool;
      lx_Start_TON_Wait : Bool;
      lx_Start_Positioning_m : Bool;
      lx_Start_FinalPositioning_m : Bool;
      lx_Start_TON_State : Bool;
      lt_TON_Wait : Time;
      ldt_MQTT : Date_And_Time;
      li_Return_LDT : Int;
      li_Lights : Int;
      li_Lights_old : Int;
      lx_State_activ : Bool;
      li_StepCase : Int;
      li_Counter : Int;
      ldi_Pos_SLD_X : DInt;
      ldi_Pos_SLD_Y : DInt;
      ldi_Pos_SLD_Z : DInt;
      ldi_Pos_Horizontal : DInt;
      ldi_Pos_Vertical : DInt;
      ldi_Pos_Rotate : DInt;
      ldi_Offset_Vertical : DInt;
      ls_Color : String;
      ls_Target : String;
      lfb_TON_Wait : TON_TIME;
      lfb_TON_State : TON_TIME;
      lfb_R_Trig_Deaktivate : R_TRIG;
      lfb_R_Trig_NiO : R_TRIG;
   END_VAR
BEGIN
   IF #lx_Init THEN

       // FB TON Wait
       #lfb_TON_Wait(IN := #lx_Start_TON_Wait,
                     PT := #lt_TON_Wait);

       #lfb_R_Trig_Deaktivate(CLK := NOT "gtyp_Setup".x_Set_Pos_Activ
                              OR NOT (("gtyp_Setup".i_Pos_Selection > 40)
                              AND ("gtyp_Setup".i_Pos_Selection < 61)));
       // Deaktivate step 150   
       IF #lfb_R_Trig_Deaktivate.Q THEN
           "gtyp_VGR".horizontal_Axis.x_Start_Positioning := FALSE;
           "gtyp_VGR".vertical_Axis.x_Start_Positioning := FALSE;
           "gtyp_VGR".rotate_Axis.x_Start_Positioning := FALSE;
           "gtyp_VGR".horizontal_Axis.x_Reference := FALSE;
           "gtyp_VGR".vertical_Axis.x_Reference := FALSE;
           "gtyp_VGR".rotate_Axis.x_Reference := FALSE;
           "gtyp_Setup".x_Start_Positioning := FALSE;
           "gtyp_Setup".x_Final_Positioning := FALSE;
           "gtyp_Setup".x_Home_Positioning := FALSE;
           "gtyp_Setup".x_Start_Offset := FALSE;
           IF (#li_StepCase > 10) THEN
               #li_StepCase := 150;
           END_IF;
       END_IF;

       // Set Positioning activ?
       IF "gtyp_Setup".x_Set_Pos_Activ
           AND (("gtyp_Setup".i_Pos_Selection > 40)
           AND ("gtyp_Setup".i_Pos_Selection < 61))
           AND ((#li_StepCase = 80)
           OR (#li_StepCase = 120)
           OR (#li_StepCase = 140)) THEN

           // Deciding which Position
           // Position - Color 
           IF "gtyp_Setup".i_Pos_Selection = 41 THEN
               #ldi_Pos_Horizontal := "gtyp_VGR".di_Pos_Color_horizontal;
               #ldi_Pos_Vertical := "gtyp_VGR".di_Pos_Color_vertical;
               #ldi_Pos_Rotate := "gtyp_VGR".di_Pos_Color_rotate;
               #ldi_Offset_Vertical := "gtyp_VGR".di_Offset_Pos_DSI_NFC_vertical;
               // Position - DSI Collect
           ELSIF "gtyp_Setup".i_Pos_Selection = 42 THEN
               #ldi_Pos_Horizontal := "gtyp_VGR".di_Pos_DSI_horizontal;
               #ldi_Pos_Vertical := "gtyp_VGR".di_Pos_DSI_Collect_vertical;
               #ldi_Pos_Rotate := "gtyp_VGR".di_Pos_DSI_rotate;
               #ldi_Offset_Vertical := "gtyp_VGR".di_Offset_Pos_DSI_NFC_vertical;
               // Position - DSI Discard 
           ELSIF "gtyp_Setup".i_Pos_Selection = 43 THEN
               #ldi_Pos_Horizontal := "gtyp_VGR".di_Pos_DSI_horizontal;
               #ldi_Pos_Vertical := "gtyp_VGR".di_Pos_DSI_Discard_vertical;
               #ldi_Pos_Rotate := "gtyp_VGR".di_Pos_DSI_rotate;
               #ldi_Offset_Vertical := "gtyp_VGR".di_Offset_Pos_DSI_NFC_vertical;
               // Position - DSO Collect 
           ELSIF "gtyp_Setup".i_Pos_Selection = 44 THEN
               #ldi_Pos_Horizontal := "gtyp_VGR".di_Pos_DSO_horizontal;
               #ldi_Pos_Vertical := "gtyp_VGR".di_Pos_DSO_Collect_vertical;
               #ldi_Pos_Rotate := "gtyp_VGR".di_Pos_DSO_rotate;
               #ldi_Offset_Vertical := "gtyp_VGR".di_Offset_Pos_DSO_vertical;
               // Position - DSO Discard 
           ELSIF "gtyp_Setup".i_Pos_Selection = 45 THEN
               #ldi_Pos_Horizontal := "gtyp_VGR".di_Pos_DSO_horizontal;
               #ldi_Pos_Vertical := "gtyp_VGR".di_Pos_DSO_Discard_vertical;
               #ldi_Pos_Rotate := "gtyp_VGR".di_Pos_DSO_rotate;
               #ldi_Offset_Vertical := "gtyp_VGR".di_Offset_Pos_DSO_vertical;
               // Position - HBW Collect 
           ELSIF "gtyp_Setup".i_Pos_Selection = 46 THEN
               #ldi_Pos_Horizontal := "gtyp_VGR".di_Pos_HBW_horizontal;
               #ldi_Pos_Vertical := "gtyp_VGR".di_Pos_HBW_Collect_vertical;
               #ldi_Pos_Rotate := "gtyp_VGR".di_Pos_HBW_rotate;
               #ldi_Offset_Vertical := "gtyp_VGR".di_Offset_Pos_HBW_vertical;
               // Position - HBW Discard 
           ELSIF "gtyp_Setup".i_Pos_Selection = 47 THEN
               #ldi_Pos_Horizontal := "gtyp_VGR".di_Pos_HBW_horizontal;
               #ldi_Pos_Vertical := "gtyp_VGR".di_Pos_HBW_Discard_vertical;
               #ldi_Pos_Rotate := "gtyp_VGR".di_Pos_HBW_rotate;
               #ldi_Offset_Vertical := "gtyp_VGR".di_Offset_Pos_HBW_vertical;
               // Position - MPO 
           ELSIF "gtyp_Setup".i_Pos_Selection = 48 THEN
               #ldi_Pos_Horizontal := "gtyp_VGR".di_Pos_MPO_horizontal;
               #ldi_Pos_Vertical := "gtyp_VGR".di_Pos_MPO_vertical;
               #ldi_Pos_Rotate := "gtyp_VGR".di_Pos_MPO_rotate;
               #ldi_Offset_Vertical := "gtyp_VGR".di_Offset_Pos_MPO_vertical;
               // Position - NFC 
           ELSIF "gtyp_Setup".i_Pos_Selection = 49 THEN
               #ldi_Pos_Horizontal := "gtyp_VGR".di_Pos_NFC_horizontal;
               #ldi_Pos_Vertical := "gtyp_VGR".di_Pos_NFC_vertical;
               #ldi_Pos_Rotate := "gtyp_VGR".di_Pos_NFC_rotate;
               #ldi_Offset_Vertical := "gtyp_VGR".di_Offset_Pos_DSI_NFC_vertical;
               // Position - NiO 
           ELSIF "gtyp_Setup".i_Pos_Selection = 50 THEN
               #ldi_Pos_Horizontal := "gtyp_VGR".di_Pos_NiO_horizontal;
               #ldi_Pos_Vertical := "gtyp_VGR".di_Pos_NiO_vertical;
               #ldi_Pos_Rotate := "gtyp_VGR".di_Pos_NiO_rotate;
               #ldi_Offset_Vertical := 500;
               // Position - SLD Blue 
           ELSIF "gtyp_Setup".i_Pos_Selection = 51 THEN
               #ldi_Pos_Horizontal := "gtyp_VGR".di_Pos_SLD_Blue_horizontal;
               #ldi_Pos_Vertical := "gtyp_VGR".di_Pos_SLD_Blue_vertical;
               #ldi_Pos_Rotate := "gtyp_VGR".di_Pos_SLD_Blue_rotate;
               #ldi_Offset_Vertical := 500;
               // Position - SLD Red 
           ELSIF "gtyp_Setup".i_Pos_Selection = 52 THEN
               #ldi_Pos_Horizontal := "gtyp_VGR".di_Pos_SLD_Red_horizontal;
               #ldi_Pos_Vertical := "gtyp_VGR".di_Pos_SLD_Red_vertical;
               #ldi_Pos_Rotate := "gtyp_VGR".di_Pos_SLD_Red_rotate;
               #ldi_Offset_Vertical := 500;
               // Position - SLD White 
           ELSIF "gtyp_Setup".i_Pos_Selection = 53 THEN
               #ldi_Pos_Horizontal := "gtyp_VGR".di_Pos_SLD_White_horizontal;
               #ldi_Pos_Vertical := "gtyp_VGR".di_Pos_SLD_White_vertical;
               #ldi_Pos_Rotate := "gtyp_VGR".di_Pos_SLD_White_rotate;
               #ldi_Offset_Vertical := 500;
           END_IF;
       END_IF;

       // Set Positioning activ?
       IF NOT "gtyp_Setup".x_Set_Pos_Activ THEN
           "gtyp_Setup".i_Pos_Selection := 0;
       END_IF;

       // step chain VGR
       CASE #li_StepCase OF

           0:  // init
               #lx_Start_TON_Wait := FALSE;
               #li_StepCase := 10;

           10:  // Set Positioning activ?
               IF "gtyp_Setup".x_Set_Pos_Activ
                   AND (("gtyp_Setup".i_Pos_Selection > 40)
                   AND ("gtyp_Setup".i_Pos_Selection < 61)) THEN

                   "gtyp_VGR".horizontal_Axis.x_Start_Positioning := FALSE;
                   "gtyp_VGR".vertical_Axis.x_Start_Positioning := FALSE;
                   "gtyp_VGR".rotate_Axis.x_Start_Positioning := FALSE;
                   "gtyp_VGR".horizontal_Axis.x_Reference := FALSE;
                   "gtyp_VGR".vertical_Axis.x_Reference := FALSE;
                   "gtyp_VGR".rotate_Axis.x_Reference := FALSE;
                   "gtyp_Setup".x_Start_Positioning := FALSE;
                   "gtyp_Setup".x_Final_Positioning := FALSE;
                   "gtyp_Setup".x_Home_Positioning := FALSE;
                   "gtyp_Setup".x_Start_Offset := FALSE;
                   "gtyp_VGR".vertical_Axis.i_PWM := 800;
                   #li_StepCase := 20;
               END_IF;

           20: // homing vertical axis
               "gtyp_VGR".vertical_Axis.x_Reference := TRUE;

               IF NOT "gtyp_VGR".vertical_Axis.x_Referenced THEN
                   #li_StepCase := 30;
               END_IF;

           30: // homed vertical axis
               IF "gtyp_VGR".vertical_Axis.x_Referenced THEN
                   "gtyp_VGR".vertical_Axis.x_Reference := FALSE;
                   #li_StepCase := 40;
               END_IF;

           40: // homing horizontal axis
               "gtyp_VGR".horizontal_Axis.x_Reference := TRUE;

               IF NOT "gtyp_VGR".horizontal_Axis.x_Referenced THEN
                   #li_StepCase := 50;
               END_IF;

           50: // homed horizontal axis
               IF "gtyp_VGR".horizontal_Axis.x_Referenced THEN
                   "gtyp_VGR".horizontal_Axis.x_Reference := FALSE;
                   #li_StepCase := 60;
               END_IF;

           60: // homing rotate axis
               "gtyp_VGR".rotate_Axis.x_Reference := TRUE;

               IF NOT "gtyp_VGR".rotate_Axis.x_Referenced THEN
                   #li_StepCase := 70;
               END_IF;

           70: // homed rotate axis
               IF "gtyp_VGR".rotate_Axis.x_Referenced THEN
                   "gtyp_VGR".rotate_Axis.x_Reference := FALSE;
                   #li_StepCase := 80;
               END_IF;

           80:  // Start Positioning Step next
               IF "gtyp_Setup".x_Start_Positioning OR #lx_Start_Positioning_m OR #lx_Start_FinalPositioning_m THEN
                   #lx_Start_Positioning_m := FALSE;
                   #li_StepCase := 90;
               END_IF;

           90: // Position rotate Axis
               "gtyp_VGR".rotate_Axis.di_Target_Position := #ldi_Pos_Rotate;
               "gtyp_VGR".rotate_Axis.x_Start_Positioning := TRUE;

               IF ("gtyp_VGR".rotate_Axis.di_Actual_Position <= (#ldi_Pos_Rotate + "gtyp_VGR".rotate_Axis.Config.di_Pos_Window))
                   AND ("gtyp_VGR".rotate_Axis.di_Actual_Position >= (#ldi_Pos_Rotate - "gtyp_VGR".rotate_Axis.Config.di_Pos_Window))
                   AND "gtyp_VGR".rotate_Axis.x_Position_Reached THEN
                   "gtyp_VGR".rotate_Axis.x_Start_Positioning := FALSE;
                   #li_StepCase := 100;
               END_IF;

           100: // Position horizontal Axis
               "gtyp_VGR".horizontal_Axis.di_Target_Position := #ldi_Pos_Horizontal;
               "gtyp_VGR".horizontal_Axis.x_Start_Positioning := TRUE;

               IF ("gtyp_VGR".horizontal_Axis.di_Actual_Position <= (#ldi_Pos_Horizontal + "gtyp_VGR".horizontal_Axis.Config.di_Pos_Window))
                   AND ("gtyp_VGR".horizontal_Axis.di_Actual_Position >= (#ldi_Pos_Horizontal - "gtyp_VGR".horizontal_Axis.Config.di_Pos_Window))
                   AND "gtyp_VGR".horizontal_Axis.x_Position_Reached THEN
                   "gtyp_VGR".horizontal_Axis.x_Start_Positioning := FALSE;
                   #li_StepCase := 110;
               END_IF;

           110: // Position vertical Axis + Offset
               "gtyp_VGR".vertical_Axis.i_PWM := 500;
               "gtyp_VGR".vertical_Axis.di_Target_Position := #ldi_Pos_Vertical - #ldi_Offset_Vertical;
               "gtyp_VGR".vertical_Axis.x_Start_Positioning := TRUE;

               IF ("gtyp_VGR".vertical_Axis.di_Actual_Position <= (#ldi_Pos_Vertical - #ldi_Offset_Vertical + "gtyp_VGR".vertical_Axis.Config.di_Pos_Window))
                   AND ("gtyp_VGR".vertical_Axis.di_Actual_Position >= (#ldi_Pos_Vertical - #ldi_Offset_Vertical - "gtyp_VGR".vertical_Axis.Config.di_Pos_Window))
                   AND "gtyp_VGR".vertical_Axis.x_Position_Reached THEN
                   "gtyp_VGR".vertical_Axis.x_Start_Positioning := FALSE;
                   "gtyp_Setup".x_Start_Positioning := FALSE;
                   #li_StepCase := 120;
               END_IF;

           120: // Deciding which doing

               // Start new Positioning
               IF "gtyp_Setup".x_Start_Positioning THEN
                   #lx_Start_Positioning_m := TRUE;
                   #li_StepCase := 10;
                   // Start Final Positioning
               ELSIF "gtyp_Setup".x_Final_Positioning OR #lx_Start_FinalPositioning_m THEN
                   #lx_Start_FinalPositioning_m := FALSE;
                   #li_StepCase := 130;
                   // Deaktivate Set Positioning
               ELSIF #lfb_R_Trig_Deaktivate.Q OR "gtyp_Setup".x_Home_Positioning THEN
                   "gtyp_Setup".x_Home_Positioning := FALSE;
                   #li_StepCase := 150;
               END_IF;

           130: // Position vertical Axis
               "gtyp_VGR".vertical_Axis.di_Target_Position := #ldi_Pos_Vertical;
               "gtyp_VGR".vertical_Axis.x_Start_Positioning := TRUE;

               IF ("gtyp_VGR".vertical_Axis.di_Actual_Position <= (#ldi_Pos_Vertical + "gtyp_VGR".vertical_Axis.Config.di_Pos_Window))
                   AND ("gtyp_VGR".vertical_Axis.di_Actual_Position >= (#ldi_Pos_Vertical - "gtyp_VGR".vertical_Axis.Config.di_Pos_Window))
                   AND "gtyp_VGR".vertical_Axis.x_Position_Reached THEN
                   "gtyp_VGR".vertical_Axis.x_Start_Positioning := FALSE;
                   "gtyp_Setup".x_Final_Positioning := FALSE;
                   #li_StepCase := 140;
               END_IF;

           140: // Deciding which doing

               // Start new Positioning
               IF "gtyp_Setup".x_Start_Positioning THEN
                   #lx_Start_Positioning_m := TRUE;
                   #li_StepCase := 10;
                   // Start Final Positioning
               ELSIF "gtyp_Setup".x_Final_Positioning THEN
                   #lx_Start_FinalPositioning_m := TRUE;
                   #li_StepCase := 10;
                   // Start Final Positioning
               ELSIF #lfb_R_Trig_Deaktivate.Q OR "gtyp_Setup".x_Home_Positioning THEN
                   "gtyp_Setup".x_Home_Positioning := FALSE;
                   #li_StepCase := 150;
               END_IF;

           150: // homing vertical axis
               "gtyp_VGR".vertical_Axis.i_PWM := 800;
               "gtyp_VGR".vertical_Axis.x_Reference := TRUE;

               IF NOT "gtyp_VGR".vertical_Axis.x_Referenced THEN
                   #li_StepCase := 160;
               END_IF;

           160: // homed vertical axis
               IF "gtyp_VGR".vertical_Axis.x_Referenced THEN
                   "gtyp_VGR".vertical_Axis.x_Reference := FALSE;
                   #li_StepCase := 170;
               END_IF;

           170: // homing horizontal axis
               "gtyp_VGR".horizontal_Axis.x_Reference := TRUE;

               IF NOT "gtyp_VGR".horizontal_Axis.x_Referenced THEN
                   #li_StepCase := 180;
               END_IF;

           180: // homed horizontal axis
               IF "gtyp_VGR".horizontal_Axis.x_Referenced THEN
                   "gtyp_VGR".horizontal_Axis.x_Reference := FALSE;
                   #li_StepCase := 0;
               END_IF;

               // Statement section ELSE    
           ELSE
               ;
       END_CASE;

       IF (("gtyp_Setup".i_Pos_Selection > 40)
           AND ("gtyp_Setup".i_Pos_Selection < 61)) THEN
           // Reload Pos Value
           "gtyp_Setup".di_Pos_Horizontal := #ldi_Pos_Horizontal;
           "gtyp_Setup".di_Pos_Vertical := #ldi_Pos_Vertical;
           "gtyp_Setup".di_Pos_Rotate := #ldi_Pos_Rotate;
       END_IF;
   ELSE
       #lx_Init := TRUE;
   END_IF;
END_FUNCTION_BLOCK

FUNCTION_BLOCK "PRG_SSC_Axis_Vertical"   // FB11, SCL
TITLE = Program Axis vertical SSC
{ S7_Optimized_Access := 'TRUE' }
AUTHOR : A.Schaefer
VERSION : 0.0
   VAR
      lx_Init : Bool;
      lfb_Vertical_Axis : "FB_Axis";
   END_VAR
BEGIN
   IF #lx_Init THEN

       // FB Axis vertical
       #lfb_Vertical_Axis(ini_Axis := 5,
                          indi_Increment := "gtyp_SSC".Vertical_Axis.di_Increment,
                          inx_Ref_Switch := "IX_SSC_RefSwitchVerticalAxis_I1",
                          inx_Referencing := "gtyp_SSC".Vertical_Axis.x_Reference,
                          inx_Start_Positioning := "gtyp_SSC".Vertical_Axis.x_Start_Positioning,
                          indi_Target_Position := "gtyp_SSC".Vertical_Axis.di_Target_Position,
                          ini_PWM := "gtyp_SSC".Vertical_Axis.i_PWM,
                          inouttyp_Config := "gtyp_SSC".Vertical_Axis.Config,
                          inouttyp_Setup := "gtyp_SetupAxis");

       "QX_SSC_M1_VerticalAxisUp_Q1" := #lfb_Vertical_Axis.outx_Motor_Pos;
       "QX_SSC_M1_VerticalAxisDown_Q2" := #lfb_Vertical_Axis.outx_Motor_Neg;
       "QW_SSC_PWM_Vertical_M1" := #lfb_Vertical_Axis.outi_Motor_PWM;
       "gtyp_SSC".Vertical_Axis.di_Actual_Position := #lfb_Vertical_Axis.outdi_Actual_Position;
       "gtyp_SSC".Vertical_Axis.x_Referenced := #lfb_Vertical_Axis.outx_Referenced;
       "gtyp_SSC".Vertical_Axis.x_Position_Reached := #lfb_Vertical_Axis.outx_Position_Reached;
   ELSE
       #lx_Init := TRUE;
   END_IF;
END_FUNCTION_BLOCK

FUNCTION_BLOCK "PRG_SSC_Ablauf"   // FB12, SCL
TITLE = Program Ablauf SSC
{ S7_Optimized_Access := 'TRUE' }
AUTHOR : A.Schaefer
VERSION : 0.0
   VAR
      lx_Init : Bool;
      lx_FirstCentre : Bool;
      lx_Start : Bool;
      lx_Start_TON_State : Bool;
      lt_TON_Wait : Time;
      li_StepCase : Int;
      ldi_TargetPosition_Horizontal : DInt;
      ldi_TargetPosition_Vertical : DInt;
      lldt_ts_old : LDT;
      ldt_write : Date_And_Time;
      li_Return_write : Int;
      ldt_MQTT : Date_And_Time;
      li_Return_LDT : Int;
      lx_Start_TON_Wait : Bool;
      ldi_StepHorizontal : DInt;
      ldi_StepVertical : DInt;
      lfb_TON_Wait : TON_TIME;
      lfb_TON_State : TON_TIME;
      lfb_F_TRIG_Set_Pos : F_TRIG;
   END_VAR
BEGIN
   IF #lx_Init THEN

       // Restart after set Positioning
       IF "gtyp_Setup".x_Set_Pos_Activ OR "gtyp_SSC".x_Start_Park_Position THEN
           #li_StepCase := 0;
       END_IF;

       // falling edge Set Pos
       #lfb_F_TRIG_Set_Pos(CLK := "gtyp_Setup".x_Set_Pos_Activ);

       IF #lfb_F_TRIG_Set_Pos.Q THEN
           #lx_FirstCentre := TRUE;
       END_IF;

       #lfb_TON_Wait(IN := #lx_Start_TON_Wait,
                     PT := #lt_TON_Wait);

       // wait time state
       #lfb_TON_State(IN := NOT #lx_Start_TON_State,
                      PT := T#2s);

       // state of the ssc cyclically transmitted to the cloud
       IF #lfb_TON_State.Q AND NOT #lx_Start_TON_State THEN
           #lx_Start_TON_State := TRUE;
           #li_Return_LDT := RD_SYS_T(#ldt_MQTT);
           "gtyp_Interface_Dashboard".Subscribe.PosPanTiltUnit.ldt_ts := DT_TO_LDT(#ldt_MQTT);
       END_IF;

       // restart wait time state
       IF NOT #lfb_TON_State.Q AND #lx_Start_TON_State THEN
           #lx_Start_TON_State := FALSE;
       END_IF;

       CASE #li_StepCase OF

           0:  // Init
               #lx_Start_TON_State := FALSE;
               "gtyp_SSC".Horizontal_Axis.x_Start_Positioning := FALSE;
               "gtyp_SSC".Vertical_Axis.x_Start_Positioning := FALSE;

               IF NOT "gtyp_Setup".x_Set_Pos_Activ AND NOT "gtyp_SSC".x_Start_Park_Position THEN
                   #li_StepCase := 10;
               END_IF;

           10: // Deciding which route to take 

               IF ("gtyp_Interface_Dashboard".Publish.PosPanTiltUnit.ldt_ts > #lldt_ts_old) OR #lx_FirstCentre THEN

                   #lldt_ts_old := "gtyp_Interface_Dashboard".Publish.PosPanTiltUnit.ldt_ts;

                   // convert the degrees to position
                   #ldi_StepHorizontal := REAL_TO_DINT("FC_Scale_linear"(inr_Y1 := DINT_TO_REAL("gtyp_SSC".Horizontal_Axis.Config.di_Neg_Soft_Switch),
                                                                                                             inr_Y2 := DINT_TO_REAL("gtyp_SSC".Horizontal_Axis.Config.di_Pos_Soft_Switch),
                                                                                                             inr_X1 := 0.0,
                                                                                                             inr_X2 := 180.0,
                                                                                                             inr_X := DINT_TO_REAL("gtyp_Interface_Dashboard".Publish.PosPanTiltUnit.i_degree)));
                   #ldi_StepVertical := REAL_TO_DINT("FC_Scale_linear"(inr_Y1 := DINT_TO_REAL("gtyp_SSC".Vertical_Axis.Config.di_Neg_Soft_Switch),
                                                                                                         inr_Y2 := DINT_TO_REAL("gtyp_SSC".Vertical_Axis.Config.di_Pos_Soft_Switch),
                                                                                                         inr_X1 := 0.0,
                                                                                                         inr_X2 := 180.0,
                                                                                                         inr_X := DINT_TO_REAL("gtyp_Interface_Dashboard".Publish.PosPanTiltUnit.i_degree)));
                   // Procedure - relmove_left
                   IF ("gtyp_Interface_Dashboard".Publish.PosPanTiltUnit.s_cmd = 'relmove_left')
                       AND (("gtyp_SSC".Horizontal_Axis.di_Actual_Position - #ldi_StepHorizontal) > "gtyp_SSC".Horizontal_Axis.Config.di_Neg_Soft_Switch + 15)
                       AND NOT "IX_SSC_RefSwitchHorizontalAxis_I2" THEN
                       #ldi_TargetPosition_Horizontal := "gtyp_SSC".Horizontal_Axis.di_Actual_Position - #ldi_StepHorizontal;
                       "gtyp_SSC".Horizontal_Axis.di_Target_Position := #ldi_TargetPosition_Horizontal;
                       "gtyp_SSC".Horizontal_Axis.x_Start_Positioning := TRUE;
                       #li_StepCase := 70;
                       // Procedure - relmove_right
                   ELSIF ("gtyp_Interface_Dashboard".Publish.PosPanTiltUnit.s_cmd = 'relmove_right')
                       AND (("gtyp_SSC".Horizontal_Axis.di_Actual_Position + #ldi_StepHorizontal) < "gtyp_SSC".Horizontal_Axis.Config.di_Pos_Soft_Switch - 15) THEN
                       #ldi_TargetPosition_Horizontal := "gtyp_SSC".Horizontal_Axis.di_Actual_Position + #ldi_StepHorizontal;
                       "gtyp_SSC".Horizontal_Axis.di_Target_Position := #ldi_TargetPosition_Horizontal;
                       "gtyp_SSC".Horizontal_Axis.x_Start_Positioning := TRUE;
                       #li_StepCase := 70;
                       // Procedure - relmove_up
                   ELSIF ("gtyp_Interface_Dashboard".Publish.PosPanTiltUnit.s_cmd = 'relmove_up')
                       AND (("gtyp_SSC".Vertical_Axis.di_Actual_Position + #ldi_StepHorizontal) < "gtyp_SSC".Vertical_Axis.Config.di_Pos_Soft_Switch - 15) THEN
                       #ldi_TargetPosition_Vertical := "gtyp_SSC".Vertical_Axis.di_Actual_Position + #ldi_StepVertical;
                       "gtyp_SSC".Vertical_Axis.di_Target_Position := #ldi_TargetPosition_Vertical;
                       "gtyp_SSC".Vertical_Axis.x_Start_Positioning := TRUE;
                       #li_StepCase := 80;
                       // Procedure - relmove_down
                   ELSIF ("gtyp_Interface_Dashboard".Publish.PosPanTiltUnit.s_cmd = 'relmove_down')
                       AND (("gtyp_SSC".Vertical_Axis.di_Actual_Position - #ldi_StepVertical) > "gtyp_SSC".Vertical_Axis.Config.di_Neg_Soft_Switch + 15)
                       AND NOT "IX_SSC_RefSwitchVerticalAxis_I1" THEN
                       #ldi_TargetPosition_Vertical := "gtyp_SSC".Vertical_Axis.di_Actual_Position - #ldi_StepVertical;
                       "gtyp_SSC".Vertical_Axis.di_Target_Position := #ldi_TargetPosition_Vertical;
                       "gtyp_SSC".Vertical_Axis.x_Start_Positioning := TRUE;
                       #li_StepCase := 80;
                       // Procedure - first 
                   ELSIF #lx_FirstCentre THEN
                       #li_StepCase := 20;
                       // Procedure - home
                   ELSIF ("gtyp_Interface_Dashboard".Publish.PosPanTiltUnit.s_cmd = 'home') THEN
                       #li_StepCase := 60;
                       // Procedure - start_pan
                   ELSIF ("gtyp_Interface_Dashboard".Publish.PosPanTiltUnit.s_cmd = 'start_pan')
                       AND ("gtyp_SSC".Horizontal_Axis.di_Actual_Position > "gtyp_SSC".Horizontal_Axis.Config.di_Neg_Soft_Switch + 15)
                       AND NOT "IX_SSC_RefSwitchHorizontalAxis_I2" THEN
                       #ldi_TargetPosition_Horizontal := "gtyp_SSC".Horizontal_Axis.Config.di_Neg_Soft_Switch + 15;
                       "gtyp_SSC".Horizontal_Axis.di_Target_Position := #ldi_TargetPosition_Horizontal;
                       "gtyp_SSC".Horizontal_Axis.x_Start_Positioning := TRUE;
                       #li_StepCase := 70;
                       // Procedure - end_pan
                   ELSIF ("gtyp_Interface_Dashboard".Publish.PosPanTiltUnit.s_cmd = 'end_pan')
                       AND ("gtyp_SSC".Horizontal_Axis.di_Actual_Position < "gtyp_SSC".Horizontal_Axis.Config.di_Pos_Soft_Switch - 15) THEN
                       #ldi_TargetPosition_Horizontal := "gtyp_SSC".Horizontal_Axis.Config.di_Pos_Soft_Switch - 15;
                       "gtyp_SSC".Horizontal_Axis.di_Target_Position := #ldi_TargetPosition_Horizontal;
                       "gtyp_SSC".Horizontal_Axis.x_Start_Positioning := TRUE;
                       #li_StepCase := 70;
                       // Procedure - start_tilt
                   ELSIF ("gtyp_Interface_Dashboard".Publish.PosPanTiltUnit.s_cmd = 'start_tilt')
                       AND ("gtyp_SSC".Vertical_Axis.di_Actual_Position > "gtyp_SSC".Vertical_Axis.Config.di_Neg_Soft_Switch + 15)
                       AND NOT "IX_SSC_RefSwitchVerticalAxis_I1" THEN
                       #ldi_TargetPosition_Vertical := "gtyp_SSC".Vertical_Axis.Config.di_Neg_Soft_Switch + 15;
                       "gtyp_SSC".Vertical_Axis.di_Target_Position := #ldi_TargetPosition_Vertical;
                       "gtyp_SSC".Vertical_Axis.x_Start_Positioning := TRUE;
                       #li_StepCase := 80;
                       // Procedure - end_tilt
                   ELSIF ("gtyp_Interface_Dashboard".Publish.PosPanTiltUnit.s_cmd = 'end_tilt')
                       AND ("gtyp_SSC".Vertical_Axis.di_Actual_Position < "gtyp_SSC".Vertical_Axis.Config.di_Pos_Soft_Switch - 15) THEN
                       #ldi_TargetPosition_Vertical := "gtyp_SSC".Vertical_Axis.Config.di_Pos_Soft_Switch - 15;
                       "gtyp_SSC".Vertical_Axis.di_Target_Position := #ldi_TargetPosition_Vertical;
                       "gtyp_SSC".Vertical_Axis.x_Start_Positioning := TRUE;
                       #li_StepCase := 80;
                   END_IF;
               END_IF;

           20: // homing vertical/horizontal axis
               "gtyp_SSC".Horizontal_Axis.x_Reference := TRUE;
               "gtyp_SSC".Vertical_Axis.x_Reference := TRUE;

               IF NOT "gtyp_SSC".Horizontal_Axis.x_Referenced AND NOT "gtyp_SSC".Vertical_Axis.x_Referenced THEN
                   #li_StepCase := 30;
               END_IF;

           30: // homed vertical/horizontal axis
               IF "gtyp_SSC".Horizontal_Axis.x_Referenced THEN
                   "gtyp_SSC".Horizontal_Axis.x_Reference := FALSE;
               END_IF;
               IF "gtyp_SSC".Vertical_Axis.x_Referenced THEN
                   "gtyp_SSC".Vertical_Axis.x_Reference := FALSE;
               END_IF;

               IF "gtyp_SSC".Horizontal_Axis.x_Referenced AND "gtyp_SSC".Vertical_Axis.x_Referenced THEN
                   "gtyp_SSC".Horizontal_Axis.x_Reference := FALSE;
                   "gtyp_SSC".Vertical_Axis.x_Reference := FALSE;
                   #lx_Start_TON_Wait := TRUE;
                   #li_StepCase := 40;
               END_IF;

           40: // wait sequence
               IF #lfb_TON_Wait.Q THEN
                   #lx_Start_TON_Wait := FALSE;
                   #li_StepCase := 50;
               END_IF;

           50: // Position horizontal/vertical axis and reached
               "gtyp_SSC".Horizontal_Axis.di_Target_Position := "gtyp_SSC".di_Pos_HBW_Horizontal;
               "gtyp_SSC".Horizontal_Axis.x_Start_Positioning := TRUE;
               "gtyp_SSC".Vertical_Axis.di_Target_Position := "gtyp_SSC".di_Pos_HBW_Vertical;
               "gtyp_SSC".Vertical_Axis.x_Start_Positioning := TRUE;

               IF ("gtyp_SSC".Horizontal_Axis.di_Actual_Position <= ("gtyp_SSC".di_Pos_HBW_Horizontal + "gtyp_SSC".Horizontal_Axis.Config.di_Pos_Window))
                   AND ("gtyp_SSC".Horizontal_Axis.di_Actual_Position >= ("gtyp_SSC".di_Pos_HBW_Horizontal - "gtyp_SSC".Horizontal_Axis.Config.di_Pos_Window))
                   AND "gtyp_SSC".Horizontal_Axis.x_Position_Reached THEN
                   "gtyp_SSC".Horizontal_Axis.x_Start_Positioning := FALSE;
               END_IF;

               IF ("gtyp_SSC".Vertical_Axis.di_Actual_Position <= ("gtyp_SSC".di_Pos_HBW_Vertical + "gtyp_SSC".Vertical_Axis.Config.di_Pos_Window))
                   AND ("gtyp_SSC".Vertical_Axis.di_Actual_Position >= ("gtyp_SSC".di_Pos_HBW_Vertical - "gtyp_SSC".Vertical_Axis.Config.di_Pos_Window))
                   AND "gtyp_SSC".Vertical_Axis.x_Position_Reached THEN
                   "gtyp_SSC".Vertical_Axis.x_Start_Positioning := FALSE;
               END_IF;

               IF ("gtyp_SSC".Horizontal_Axis.di_Actual_Position <= ("gtyp_SSC".di_Pos_HBW_Horizontal + "gtyp_SSC".Horizontal_Axis.Config.di_Pos_Window))
                   AND ("gtyp_SSC".Horizontal_Axis.di_Actual_Position >= ("gtyp_SSC".di_Pos_HBW_Horizontal - "gtyp_SSC".Horizontal_Axis.Config.di_Pos_Window))
                   AND "gtyp_SSC".Horizontal_Axis.x_Position_Reached
                   AND ("gtyp_SSC".Vertical_Axis.di_Actual_Position <= ("gtyp_SSC".di_Pos_HBW_Vertical + "gtyp_SSC".Vertical_Axis.Config.di_Pos_Window))
                   AND ("gtyp_SSC".Vertical_Axis.di_Actual_Position >= ("gtyp_SSC".di_Pos_HBW_Vertical - "gtyp_SSC".Vertical_Axis.Config.di_Pos_Window))
                   AND "gtyp_SSC".Vertical_Axis.x_Position_Reached THEN
                   "gtyp_SSC".Horizontal_Axis.x_Start_Positioning := FALSE;
                   "gtyp_SSC".Vertical_Axis.x_Start_Positioning := FALSE;
                   #lx_FirstCentre := FALSE;
                   #li_StepCase := 90;
               END_IF;

           60: // Position Centre horizontal/vertical axis and reached
               "gtyp_SSC".Horizontal_Axis.di_Target_Position := "gtyp_SSC".di_Pos_Centre_Horizontal;
               "gtyp_SSC".Horizontal_Axis.x_Start_Positioning := TRUE;
               "gtyp_SSC".Vertical_Axis.di_Target_Position := "gtyp_SSC".di_Pos_Centre_Vertical;
               "gtyp_SSC".Vertical_Axis.x_Start_Positioning := TRUE;

               IF ("gtyp_SSC".Horizontal_Axis.di_Actual_Position <= ("gtyp_SSC".di_Pos_Centre_Horizontal + "gtyp_SSC".Horizontal_Axis.Config.di_Pos_Window))
                   AND ("gtyp_SSC".Horizontal_Axis.di_Actual_Position >= ("gtyp_SSC".di_Pos_Centre_Horizontal - "gtyp_SSC".Horizontal_Axis.Config.di_Pos_Window))
                   AND "gtyp_SSC".Horizontal_Axis.x_Position_Reached THEN
                   "gtyp_SSC".Horizontal_Axis.x_Start_Positioning := FALSE;
               END_IF;

               IF ("gtyp_SSC".Vertical_Axis.di_Actual_Position <= ("gtyp_SSC".di_Pos_Centre_Vertical + "gtyp_SSC".Vertical_Axis.Config.di_Pos_Window))
                   AND ("gtyp_SSC".Vertical_Axis.di_Actual_Position >= ("gtyp_SSC".di_Pos_Centre_Vertical - "gtyp_SSC".Vertical_Axis.Config.di_Pos_Window))
                   AND "gtyp_SSC".Vertical_Axis.x_Position_Reached THEN
                   "gtyp_SSC".Vertical_Axis.x_Start_Positioning := FALSE;
               END_IF;

               IF ("gtyp_SSC".Horizontal_Axis.di_Actual_Position <= ("gtyp_SSC".di_Pos_Centre_Horizontal + "gtyp_SSC".Horizontal_Axis.Config.di_Pos_Window))
                   AND ("gtyp_SSC".Horizontal_Axis.di_Actual_Position >= ("gtyp_SSC".di_Pos_Centre_Horizontal - "gtyp_SSC".Horizontal_Axis.Config.di_Pos_Window))
                   AND "gtyp_SSC".Horizontal_Axis.x_Position_Reached
                   AND ("gtyp_SSC".Vertical_Axis.di_Actual_Position <= ("gtyp_SSC".di_Pos_Centre_Vertical + "gtyp_SSC".Vertical_Axis.Config.di_Pos_Window))
                   AND ("gtyp_SSC".Vertical_Axis.di_Actual_Position >= ("gtyp_SSC".di_Pos_Centre_Vertical - "gtyp_SSC".Vertical_Axis.Config.di_Pos_Window))
                   AND "gtyp_SSC".Vertical_Axis.x_Position_Reached THEN
                   "gtyp_SSC".Horizontal_Axis.x_Start_Positioning := FALSE;
                   "gtyp_SSC".Vertical_Axis.x_Start_Positioning := FALSE;
                   #lx_FirstCentre := FALSE;
                   #li_StepCase := 90;
               END_IF;

           70: // Position horizontal axis reached
               IF ("gtyp_SSC".Horizontal_Axis.di_Actual_Position <= (#ldi_TargetPosition_Horizontal + "gtyp_SSC".Horizontal_Axis.Config.di_Pos_Window))
                   AND ("gtyp_SSC".Horizontal_Axis.di_Actual_Position >= (#ldi_TargetPosition_Horizontal - "gtyp_SSC".Horizontal_Axis.Config.di_Pos_Window))
                   AND "gtyp_SSC".Horizontal_Axis.x_Position_Reached THEN
                   "gtyp_SSC".Horizontal_Axis.x_Start_Positioning := FALSE;
                   #li_StepCase := 90;
               END_IF;

           80: // Position vertical axis reached
               IF ("gtyp_SSC".Vertical_Axis.di_Actual_Position <= (#ldi_TargetPosition_Vertical + "gtyp_SSC".Vertical_Axis.Config.di_Pos_Window))
                   AND ("gtyp_SSC".Vertical_Axis.di_Actual_Position >= (#ldi_TargetPosition_Vertical - "gtyp_SSC".Vertical_Axis.Config.di_Pos_Window))
                   AND "gtyp_SSC".Vertical_Axis.x_Position_Reached THEN
                   "gtyp_SSC".Vertical_Axis.x_Start_Positioning := FALSE;
                   #li_StepCase := 90;
               END_IF;

           90: // convert the position to degrees
               "gtyp_Interface_Dashboard".Subscribe.PosPanTiltUnit.r_pan := "FC_Scale_linear"(inr_Y1 := -1.0,
                                                                                              inr_Y2 := 1.0,
                                                                                              inr_X1 := DINT_TO_REAL("gtyp_SSC".Horizontal_Axis.Config.di_Neg_Soft_Switch),
                                                                                              inr_X2 := DINT_TO_REAL("gtyp_SSC".Horizontal_Axis.Config.di_Pos_Soft_Switch),
                                                                                              inr_X := "gtyp_SSC".Horizontal_Axis.di_Actual_Position);
               "gtyp_Interface_Dashboard".Subscribe.PosPanTiltUnit.r_tilt := "FC_Scale_linear"(inr_Y1 := -1.0,
                                                                                               inr_Y2 := 1.0,
                                                                                               inr_X1 := DINT_TO_REAL("gtyp_SSC".Vertical_Axis.Config.di_Neg_Soft_Switch),
                                                                                               inr_X2 := DINT_TO_REAL("gtyp_SSC".Vertical_Axis.Config.di_Pos_Soft_Switch),
                                                                                               inr_X := "gtyp_SSC".Vertical_Axis.di_Actual_Position);

               #li_Return_write := RD_SYS_T(#ldt_write);
               "gtyp_Interface_Dashboard".Subscribe.PosPanTiltUnit.ldt_ts := DT_TO_LDT(#ldt_write);
               #lx_Start_TON_Wait := TRUE;
               #li_StepCase := 100;

           100:// wait sequence
               IF #lfb_TON_Wait.Q THEN
                   #lx_Start_TON_Wait := FALSE;
                   #li_StepCase := 0;
               END_IF;
               // Statement section ELSE        
           ELSE
               ;
       END_CASE;

   ELSE
       #lx_Init := TRUE;
       #lx_FirstCentre := TRUE;

       "gtyp_SSC".x_Start_Park_Position := FALSE;
       "gtyp_SSC".x_Park_Position_Reached := FALSE;
       "gtyp_SSC".x_Error := FALSE;
   END_IF;
END_FUNCTION_BLOCK

FUNCTION_BLOCK "PRG_SSC_Set_Positioning"   // FB13, SCL
TITLE = Program Set Positioning SSC
{ S7_Optimized_Access := 'TRUE' }
AUTHOR : A.Schaefer
VERSION : 0.0
   VAR
      lx_Init : Bool;
      lx_Start_TON_Wait : Bool;
      lx_Start_Positioning_m : Bool;
      lt_TON_Wait : Time;
      li_StepCase : Int;
      ldi_Pos_Horizontal : DInt;
      ldi_Pos_Vertical : DInt;
      lfb_R_Trig_Deaktivate : R_TRIG;
      lfb_TON_Wait : TON_TIME;
   END_VAR
BEGIN
   IF #lx_Init THEN

       // FB TON Wait
       #lfb_TON_Wait(IN := #lx_Start_TON_Wait,
                     PT := #lt_TON_Wait);

       #lfb_R_Trig_Deaktivate(CLK := NOT "gtyp_Setup".x_Set_Pos_Activ
                              OR NOT (("gtyp_Setup".i_Pos_Selection > 0)
                              AND ("gtyp_Setup".i_Pos_Selection < 21)));
       // Deaktivate step 10   
       IF #lfb_R_Trig_Deaktivate.Q THEN
           "gtyp_SSC".Horizontal_Axis.x_Start_Positioning := FALSE;
           "gtyp_SSC".Vertical_Axis.x_Start_Positioning := FALSE;
           "gtyp_SSC".Horizontal_Axis.x_Reference := FALSE;
           "gtyp_SSC".Vertical_Axis.x_Reference := FALSE;
           "gtyp_Setup".x_Start_Positioning := FALSE;
           "gtyp_Setup".x_Final_Positioning := FALSE;
           "gtyp_Setup".x_Home_Positioning := FALSE;
           "gtyp_Setup".x_Start_Offset := FALSE;
           #lx_Start_Positioning_m := FALSE;
           IF (#li_StepCase > 10) THEN
               #li_StepCase := 70;
           END_IF;
       END_IF;

       // Set Positioning activ?
       IF "gtyp_Setup".x_Set_Pos_Activ
           AND (("gtyp_Setup".i_Pos_Selection > 0)
           AND ("gtyp_Setup".i_Pos_Selection < 21))
           AND ((#li_StepCase = 40)
           OR (#li_StepCase = 60)) THEN

           // Deciding which Position
           // Position - Centre
           IF "gtyp_Setup".i_Pos_Selection = 1 THEN
               #ldi_Pos_Horizontal := "gtyp_SSC".di_Pos_Centre_Horizontal;
               #ldi_Pos_Vertical := "gtyp_SSC".di_Pos_Centre_Vertical;
               // Position - HBW 
           ELSIF "gtyp_Setup".i_Pos_Selection = 2 THEN
               #ldi_Pos_Horizontal := "gtyp_SSC".di_Pos_HBW_Horizontal;
               #ldi_Pos_Vertical := "gtyp_SSC".di_Pos_HBW_Vertical;
           END_IF;
       END_IF;

       // Set Positioning activ?
       IF NOT "gtyp_Setup".x_Set_Pos_Activ THEN
           "gtyp_Setup".i_Pos_Selection := 0;
       END_IF;

       // step chain HBW
       CASE #li_StepCase OF

           0:  // init
               #lx_Start_TON_Wait := FALSE;
               #li_StepCase := 10;

           10:  // Set Positioning activ?
               IF "gtyp_Setup".x_Set_Pos_Activ
                   AND (("gtyp_Setup".i_Pos_Selection > 0)
                   AND ("gtyp_Setup".i_Pos_Selection < 21)) THEN
                   "gtyp_SSC".Horizontal_Axis.x_Start_Positioning := FALSE;
                   "gtyp_SSC".Vertical_Axis.x_Start_Positioning := FALSE;
                   "gtyp_SSC".Horizontal_Axis.x_Reference := FALSE;
                   "gtyp_SSC".Vertical_Axis.x_Reference := FALSE;
                   "gtyp_Setup".x_Start_Positioning := FALSE;
                   "gtyp_Setup".x_Final_Positioning := FALSE;
                   "gtyp_Setup".x_Home_Positioning := FALSE;
                   "gtyp_Setup".x_Start_Offset := FALSE;
                   #li_StepCase := 20;
               END_IF;

           20: //homing vertical/horizontal axis

               "gtyp_SSC".Horizontal_Axis.x_Reference := TRUE;
               "gtyp_SSC".Vertical_Axis.x_Reference := TRUE;

               IF NOT "gtyp_SSC".Horizontal_Axis.x_Referenced AND NOT "gtyp_SSC".Vertical_Axis.x_Referenced THEN
                   #li_StepCase := 30;
               END_IF;

           30: // homed vertical/horizontal axis
               IF "gtyp_SSC".Horizontal_Axis.x_Referenced THEN
                   "gtyp_SSC".Horizontal_Axis.x_Reference := FALSE;
               END_IF;
               IF "gtyp_SSC".Vertical_Axis.x_Referenced THEN
                   "gtyp_SSC".Vertical_Axis.x_Reference := FALSE;
               END_IF;

               IF "gtyp_SSC".Horizontal_Axis.x_Referenced AND "gtyp_SSC".Vertical_Axis.x_Referenced THEN
                   "gtyp_SSC".Horizontal_Axis.x_Reference := FALSE;
                   "gtyp_SSC".Vertical_Axis.x_Reference := FALSE;
                   #li_StepCase := 40;
               END_IF;

           40:  // Start Positioning Step next
               IF "gtyp_Setup".x_Start_Positioning OR #lx_Start_Positioning_m THEN
                   #lx_Start_Positioning_m := FALSE;
                   #li_StepCase := 50;
               END_IF;

           50: // Position vertical/horizontal HBW
               "gtyp_SSC".Horizontal_Axis.di_Target_Position := #ldi_Pos_Horizontal;
               "gtyp_SSC".Horizontal_Axis.x_Start_Positioning := TRUE;
               "gtyp_SSC".Vertical_Axis.di_Target_Position := #ldi_Pos_Vertical;
               "gtyp_SSC".Vertical_Axis.x_Start_Positioning := TRUE;

               IF ("gtyp_SSC".Horizontal_Axis.di_Actual_Position <= (#ldi_Pos_Horizontal + "gtyp_SSC".Horizontal_Axis.Config.di_Pos_Window))
                   AND ("gtyp_SSC".Horizontal_Axis.di_Actual_Position >= (#ldi_Pos_Horizontal - "gtyp_SSC".Horizontal_Axis.Config.di_Pos_Window))
                   AND "gtyp_SSC".Horizontal_Axis.x_Position_Reached THEN
                   "gtyp_SSC".Horizontal_Axis.x_Start_Positioning := FALSE;
               END_IF;

               IF ("gtyp_SSC".Vertical_Axis.di_Actual_Position <= (#ldi_Pos_Vertical + "gtyp_SSC".Vertical_Axis.Config.di_Pos_Window))
                   AND ("gtyp_SSC".Vertical_Axis.di_Actual_Position >= (#ldi_Pos_Vertical - "gtyp_SSC".Vertical_Axis.Config.di_Pos_Window))
                   AND "gtyp_SSC".Vertical_Axis.x_Position_Reached THEN
                   "gtyp_SSC".Vertical_Axis.x_Start_Positioning := FALSE;
               END_IF;

               IF ("gtyp_SSC".Horizontal_Axis.di_Actual_Position <= (#ldi_Pos_Horizontal + "gtyp_SSC".Horizontal_Axis.Config.di_Pos_Window))
                   AND ("gtyp_SSC".Horizontal_Axis.di_Actual_Position >= (#ldi_Pos_Horizontal - "gtyp_SSC".Horizontal_Axis.Config.di_Pos_Window))
                   AND "gtyp_SSC".Horizontal_Axis.x_Position_Reached
                   AND ("gtyp_SSC".Vertical_Axis.di_Actual_Position <= (#ldi_Pos_Vertical + "gtyp_SSC".Vertical_Axis.Config.di_Pos_Window))
                   AND ("gtyp_SSC".Vertical_Axis.di_Actual_Position >= (#ldi_Pos_Vertical - "gtyp_SSC".Vertical_Axis.Config.di_Pos_Window))
                   AND "gtyp_SSC".Vertical_Axis.x_Position_Reached THEN
                   "gtyp_SSC".Horizontal_Axis.x_Start_Positioning := FALSE;
                   "gtyp_SSC".Vertical_Axis.x_Start_Positioning := FALSE;
                   "gtyp_Setup".x_Start_Positioning := FALSE;
                   #li_StepCase := 60;
               END_IF;

           60: // Deciding which doing

               // Start new Positioning
               IF "gtyp_Setup".x_Start_Positioning OR "gtyp_Setup".x_Home_Positioning THEN
                   #lx_Start_Positioning_m := TRUE;
                   #li_StepCase := 10;
               ELSIF #lfb_R_Trig_Deaktivate.Q THEN
                   "gtyp_Setup".x_Home_Positioning := FALSE;
                   #li_StepCase := 70;
               END_IF;

           70: //homing vertical/horizontal axis

               "gtyp_SSC".Horizontal_Axis.x_Reference := TRUE;
               "gtyp_SSC".Vertical_Axis.x_Reference := TRUE;

               IF NOT "gtyp_SSC".Horizontal_Axis.x_Referenced AND NOT "gtyp_SSC".Vertical_Axis.x_Referenced THEN
                   #li_StepCase := 80;
               END_IF;

           80: // homed vertical/horizontal axis
               IF "gtyp_SSC".Horizontal_Axis.x_Referenced THEN
                   "gtyp_SSC".Horizontal_Axis.x_Reference := FALSE;
               END_IF;
               IF "gtyp_SSC".Vertical_Axis.x_Referenced THEN
                   "gtyp_SSC".Vertical_Axis.x_Reference := FALSE;
               END_IF;

               IF "gtyp_SSC".Horizontal_Axis.x_Referenced AND "gtyp_SSC".Vertical_Axis.x_Referenced THEN
                   "gtyp_SSC".Horizontal_Axis.x_Reference := FALSE;
                   "gtyp_SSC".Vertical_Axis.x_Reference := FALSE;
                   #li_StepCase := 0;
               END_IF;

               // Statement section ELSE    
           ELSE
               ;
       END_CASE;

       IF (("gtyp_Setup".i_Pos_Selection > 0)
           AND ("gtyp_Setup".i_Pos_Selection < 21)) THEN
           // Reload Pos Value
           "gtyp_Setup".di_Pos_Horizontal := #ldi_Pos_Horizontal;
           "gtyp_Setup".di_Pos_Vertical := #ldi_Pos_Vertical;
           "gtyp_Setup".di_Pos_Rotate := 0;
       END_IF;
   ELSE
       #lx_Init := TRUE;
   END_IF;
END_FUNCTION_BLOCK

FUNCTION_BLOCK "PRG_HBW_Axis_Horizontal"   // FB14, SCL
TITLE = Program Axis horizontal HBW
{ S7_Optimized_Access := 'TRUE' }
AUTHOR : A.Schaefer
VERSION : 0.0
   VAR
      lx_Init : Bool;
      lfb_Horizontal_Axis : "FB_Axis_Auto";
   END_VAR
BEGIN
   IF #lx_Init THEN

       // FB Axis horizontal
       #lfb_Horizontal_Axis(ini_Axis := 6,
                            indi_Increment := "gtyp_HBW".Horizontal_Axis.di_Increment,
                            inx_Ref_Switch := "IX_HBW_RefSwitchHorizontalAxis_I1",
                            inx_Referencing := "gtyp_HBW".Horizontal_Axis.x_Reference,
                            inx_Start_Positioning := "gtyp_HBW".Horizontal_Axis.x_Start_Positioning,
                            indi_Target_Position := "gtyp_HBW".Horizontal_Axis.di_Target_Position,
                            ini_PWM := "gtyp_HBW".Horizontal_Axis.i_PWM,
                            inouttyp_Config := "gtyp_HBW".Horizontal_Axis.Config,
                            inouttyp_Setup := "gtyp_SetupAxis");

       "QX_HBW_M2_HorizontalTowardsRack_Q3" := #lfb_Horizontal_Axis.outx_Motor_Pos;
       "QX_HBW_M2_HorizontalTowardsConveyorBelt_Q4" := #lfb_Horizontal_Axis.outx_Motor_Neg;
       "QW_HBW_PWM_HorizontalAxis_M2" := #lfb_Horizontal_Axis.outi_Motor_PWM;
       "gtyp_HBW".Horizontal_Axis.di_Actual_Position := #lfb_Horizontal_Axis.outdi_Actual_Position;
       "gtyp_HBW".Horizontal_Axis.x_Referenced := #lfb_Horizontal_Axis.outx_Referenced;
       "gtyp_HBW".Horizontal_Axis.x_Position_Reached := #lfb_Horizontal_Axis.outx_Position_Reached;
   ELSE
       #lx_Init := TRUE;
   END_IF;
END_FUNCTION_BLOCK

FUNCTION_BLOCK "PRG_HBW_Axis_Vertical"   // FB15, SCL
TITLE = Program Axis vertical HBW
{ S7_Optimized_Access := 'TRUE' }
AUTHOR : A.Schaefer
VERSION : 0.0
   VAR
      lx_Init : Bool;
      lfb_Vertical_Axis : "FB_Axis_Auto";
   END_VAR
BEGIN
   IF #lx_Init THEN

       // FB Axis vertical
       #lfb_Vertical_Axis(ini_Axis := 7,
                          indi_Increment := "gtyp_HBW".Vertical_Axis.di_Increment,
                          inx_Ref_Switch := "IX_HBW_RefSwitchVerticalAxis_I4",
                          inx_Referencing := "gtyp_HBW".Vertical_Axis.x_Reference,
                          inx_Start_Positioning := "gtyp_HBW".Vertical_Axis.x_Start_Positioning,
                          indi_Target_Position := "gtyp_HBW".Vertical_Axis.di_Target_Position,
                          ini_PWM := "gtyp_HBW".Vertical_Axis.i_PWM,
                          inouttyp_Config := "gtyp_HBW".Vertical_Axis.Config,
                          inouttyp_Setup := "gtyp_SetupAxis");

       "QX_HBW_M3_VerticalAxisDownward_Q5" := #lfb_Vertical_Axis.outx_Motor_Pos;
       "QX_HBW_M3_VerticalAxisUpward_Q6" := #lfb_Vertical_Axis.outx_Motor_Neg;
       "QW_HBW_PWM_VerticalAxis_M3" := #lfb_Vertical_Axis.outi_Motor_PWM;
       "gtyp_HBW".Vertical_Axis.di_Actual_Position := #lfb_Vertical_Axis.outdi_Actual_Position;
       "gtyp_HBW".Vertical_Axis.x_Referenced := #lfb_Vertical_Axis.outx_Referenced;
       "gtyp_HBW".Vertical_Axis.x_Position_Reached := #lfb_Vertical_Axis.outx_Position_Reached;
   ELSE
       #lx_Init := TRUE;
   END_IF;
END_FUNCTION_BLOCK

FUNCTION_BLOCK "PRG_HBW_Ablauf"   // FB16, SCL
TITLE = Program Ablauf HBW
{ S7_Optimized_Access := 'TRUE' }
AUTHOR : A.Schaefer
VERSION : 0.1
   VAR
      lx_Init : Bool;
      lx_Start_TON_Fill_HBW : Bool;
      lx_Start_TON_Wait : Bool;
      lx_Time_Error : Bool;
      lt_TON_Wait : Time;
      lx_Start_TON_State : Bool;
      lx_Storage : Bool;
      ldt_MQTT : Date_And_Time;
      li_Return_LDT : Int;
      lldt_Outsource : LDT;
      li_Lights : Int;
      li_Lights_old : Int;
      li_Counter_Act_Hor : Int;
      li_Counter_Act_Ver : Int;
      li_StepCase : Int;
      ldi_PosRack_Horizontal : DInt;
      ldi_PosRack_Vertical : DInt;
      ls_Color : String;
      lfb_TON_State : TON_TIME;
      lfb_TON_ConveyerBelt_Out : TON_TIME;
      lfb_TON_Wait : TON_TIME;
      lfb_TON_Fill_HBW : TON_TIME;
      lfb_TON_Error : TON_TIME;
   END_VAR
   VAR_TEMP
      ti_Counter : Int;
      ti_Counter_Hor : Int;
      ti_Counter_Ver : Int;
      tx_Found_Position : Bool;
   END_VAR
BEGIN
   IF #lx_Init THEN

       // Restart after set Positioning
       IF "gtyp_Setup".x_Set_Pos_Activ OR "gtyp_HBW".x_Start_Park_Position THEN
           #li_StepCase := 0;
       END_IF;

       // wait time state
       #lfb_TON_State(IN := NOT #lx_Start_TON_State,
                      PT := T#2s);

       // runtime monitoring error
       #lfb_TON_Error(IN := #lx_Time_Error,
                      PT := T#30s);

       // Fill the HBW-Rack with Items
       #lfb_TON_Fill_HBW(IN := #lx_Start_TON_Fill_HBW,
                         PT := T#60s);

       IF #lfb_TON_Fill_HBW.Q THEN
           #lx_Start_TON_Fill_HBW := FALSE;
       END_IF;

       IF #lx_Start_TON_Fill_HBW AND ("IX_Fill_HBW" OR "gtyp_Setup".x_Fill_Rack_HBW) THEN
           #li_Return_LDT := RD_SYS_T(#ldt_MQTT);

           "gtyp_HBW".Rack_Workpiece[1, 1].s_id := '04c34892186580';
           "gtyp_HBW".Rack_Workpiece[1, 1].s_state := 'RAW';
           "gtyp_HBW".Rack_Workpiece[1, 1].s_type := 'WHITE';
           "gtyp_HBW".Rack_History[1, 1].History[1].ldt_ts := DT_TO_LDT(#ldt_MQTT);
           "gtyp_HBW".Rack_History[1, 1].History[1].i_code := 100;
           "gtyp_HBW".Rack_History[1, 1].History[2].ldt_ts := DT_TO_LDT(#ldt_MQTT);
           "gtyp_HBW".Rack_History[1, 1].History[2].i_code := 200;
           "gtyp_HBW".Rack_History[1, 1].History[3].ldt_ts := DT_TO_LDT(#ldt_MQTT);
           "gtyp_HBW".Rack_History[1, 1].History[3].i_code := 300;

           "gtyp_HBW".Rack_Workpiece[1, 2].s_id := '04c34892186581';
           "gtyp_HBW".Rack_Workpiece[1, 2].s_state := 'RAW';
           "gtyp_HBW".Rack_Workpiece[1, 2].s_type := 'WHITE';
           "gtyp_HBW".Rack_History[1, 2].History[1].ldt_ts := DT_TO_LDT(#ldt_MQTT);
           "gtyp_HBW".Rack_History[1, 2].History[1].i_code := 100;
           "gtyp_HBW".Rack_History[1, 2].History[2].ldt_ts := DT_TO_LDT(#ldt_MQTT);
           "gtyp_HBW".Rack_History[1, 2].History[2].i_code := 200;
           "gtyp_HBW".Rack_History[1, 2].History[3].ldt_ts := DT_TO_LDT(#ldt_MQTT);
           "gtyp_HBW".Rack_History[1, 2].History[3].i_code := 300;

           "gtyp_HBW".Rack_Workpiece[1, 3].s_id := '04c34892186582';
           "gtyp_HBW".Rack_Workpiece[1, 3].s_state := 'RAW';
           "gtyp_HBW".Rack_Workpiece[1, 3].s_type := 'WHITE';
           "gtyp_HBW".Rack_History[1, 3].History[1].ldt_ts := DT_TO_LDT(#ldt_MQTT);
           "gtyp_HBW".Rack_History[1, 3].History[1].i_code := 100;
           "gtyp_HBW".Rack_History[1, 3].History[2].ldt_ts := DT_TO_LDT(#ldt_MQTT);
           "gtyp_HBW".Rack_History[1, 3].History[2].i_code := 200;
           "gtyp_HBW".Rack_History[1, 3].History[3].ldt_ts := DT_TO_LDT(#ldt_MQTT);
           "gtyp_HBW".Rack_History[1, 3].History[3].i_code := 300;

           "gtyp_HBW".Rack_Workpiece[2, 1].s_id := '04c34892186583';
           "gtyp_HBW".Rack_Workpiece[2, 1].s_state := 'RAW';
           "gtyp_HBW".Rack_Workpiece[2, 1].s_type := 'RED';
           "gtyp_HBW".Rack_History[2, 1].History[1].ldt_ts := DT_TO_LDT(#ldt_MQTT);
           "gtyp_HBW".Rack_History[2, 1].History[1].i_code := 100;
           "gtyp_HBW".Rack_History[2, 1].History[2].ldt_ts := DT_TO_LDT(#ldt_MQTT);
           "gtyp_HBW".Rack_History[2, 1].History[2].i_code := 200;
           "gtyp_HBW".Rack_History[2, 1].History[3].ldt_ts := DT_TO_LDT(#ldt_MQTT);
           "gtyp_HBW".Rack_History[2, 1].History[3].i_code := 300;

           "gtyp_HBW".Rack_Workpiece[2, 2].s_id := '04c34892186584';
           "gtyp_HBW".Rack_Workpiece[2, 2].s_state := 'RAW';
           "gtyp_HBW".Rack_Workpiece[2, 2].s_type := 'RED';
           "gtyp_HBW".Rack_History[2, 2].History[1].ldt_ts := DT_TO_LDT(#ldt_MQTT);
           "gtyp_HBW".Rack_History[2, 2].History[1].i_code := 100;
           "gtyp_HBW".Rack_History[2, 2].History[2].ldt_ts := DT_TO_LDT(#ldt_MQTT);
           "gtyp_HBW".Rack_History[2, 2].History[2].i_code := 200;
           "gtyp_HBW".Rack_History[2, 2].History[3].ldt_ts := DT_TO_LDT(#ldt_MQTT);
           "gtyp_HBW".Rack_History[2, 2].History[3].i_code := 300;

           "gtyp_HBW".Rack_Workpiece[2, 3].s_id := '04c34892186585';
           "gtyp_HBW".Rack_Workpiece[2, 3].s_state := 'RAW';
           "gtyp_HBW".Rack_Workpiece[2, 3].s_type := 'RED';
           "gtyp_HBW".Rack_History[2, 3].History[1].ldt_ts := DT_TO_LDT(#ldt_MQTT);
           "gtyp_HBW".Rack_History[2, 3].History[1].i_code := 100;
           "gtyp_HBW".Rack_History[2, 3].History[2].ldt_ts := DT_TO_LDT(#ldt_MQTT);
           "gtyp_HBW".Rack_History[2, 3].History[2].i_code := 200;
           "gtyp_HBW".Rack_History[2, 3].History[3].ldt_ts := DT_TO_LDT(#ldt_MQTT);
           "gtyp_HBW".Rack_History[2, 3].History[3].i_code := 300;

           "gtyp_HBW".Rack_Workpiece[3, 1].s_id := '04c34892186586';
           "gtyp_HBW".Rack_Workpiece[3, 1].s_state := 'RAW';
           "gtyp_HBW".Rack_Workpiece[3, 1].s_type := 'BLUE';
           "gtyp_HBW".Rack_History[3, 1].History[1].ldt_ts := DT_TO_LDT(#ldt_MQTT);
           "gtyp_HBW".Rack_History[3, 1].History[1].i_code := 100;
           "gtyp_HBW".Rack_History[3, 1].History[2].ldt_ts := DT_TO_LDT(#ldt_MQTT);
           "gtyp_HBW".Rack_History[3, 1].History[2].i_code := 200;
           "gtyp_HBW".Rack_History[3, 1].History[3].ldt_ts := DT_TO_LDT(#ldt_MQTT);
           "gtyp_HBW".Rack_History[3, 1].History[3].i_code := 300;

           "gtyp_HBW".Rack_Workpiece[3, 2].s_id := '04c34892186587';
           "gtyp_HBW".Rack_Workpiece[3, 2].s_state := 'RAW';
           "gtyp_HBW".Rack_Workpiece[3, 2].s_type := 'BLUE';
           "gtyp_HBW".Rack_History[3, 2].History[1].ldt_ts := DT_TO_LDT(#ldt_MQTT);
           "gtyp_HBW".Rack_History[3, 2].History[1].i_code := 100;
           "gtyp_HBW".Rack_History[3, 2].History[2].ldt_ts := DT_TO_LDT(#ldt_MQTT);
           "gtyp_HBW".Rack_History[3, 2].History[2].i_code := 200;
           "gtyp_HBW".Rack_History[3, 2].History[3].ldt_ts := DT_TO_LDT(#ldt_MQTT);
           "gtyp_HBW".Rack_History[3, 2].History[3].i_code := 300;

           "gtyp_HBW".Rack_Workpiece[3, 3].s_id := '04c34892186588';
           "gtyp_HBW".Rack_Workpiece[3, 3].s_state := 'RAW';
           "gtyp_HBW".Rack_Workpiece[3, 3].s_type := 'BLUE';
           "gtyp_HBW".Rack_History[3, 3].History[1].ldt_ts := DT_TO_LDT(#ldt_MQTT);
           "gtyp_HBW".Rack_History[3, 3].History[1].i_code := 100;
           "gtyp_HBW".Rack_History[3, 3].History[2].ldt_ts := DT_TO_LDT(#ldt_MQTT);
           "gtyp_HBW".Rack_History[3, 3].History[2].i_code := 200;
           "gtyp_HBW".Rack_History[3, 3].History[3].ldt_ts := DT_TO_LDT(#ldt_MQTT);
           "gtyp_HBW".Rack_History[3, 3].History[3].i_code := 300;

           #lx_Start_TON_Fill_HBW := FALSE;
           "gtyp_Setup".x_Fill_Rack_HBW := FALSE;
       END_IF;

       "gtyp_Setup".x_Start_TON_Fill_HBW := #lx_Start_TON_Fill_HBW;

       // state of the Stock HBW cyclically transmitted to the cloud
       IF (#lfb_TON_State.Q OR (#li_Lights <> #li_Lights_old)) AND NOT #lx_Start_TON_State THEN
           #li_Lights_old := #li_Lights;
           #lx_Start_TON_State := TRUE;
           #li_Return_LDT := RD_SYS_T(#ldt_MQTT);
           "gtyp_Interface_Dashboard".Subscribe.Stock_HBW.StockItem := "gtyp_HBW".Rack_Workpiece;
           "gtyp_Interface_Dashboard".Subscribe.Stock_HBW.ldt_ts := DT_TO_LDT(#ldt_MQTT);

           "gtyp_Interface_Dashboard".Subscribe.State_HBW.ldt_ts := DT_TO_LDT(#ldt_MQTT);
           "gtyp_Interface_Dashboard".Subscribe.State_HBW.i_code := #li_Lights;
           "gtyp_Interface_Dashboard".Subscribe.State_HBW.s_description := '';
           "gtyp_Interface_Dashboard".Subscribe.State_HBW.s_station := 'hbw';
           "gtyp_Interface_Dashboard".Subscribe.State_HBW.s_target := '';
       END_IF;

       // restart wait time state
       IF NOT #lfb_TON_State.Q AND #lx_Start_TON_State THEN
           #lx_Start_TON_State := FALSE;
       END_IF;

       // FB TON Wait
       #lfb_TON_Wait(IN := #lx_Start_TON_Wait,
                     PT := #lt_TON_Wait);

       //Run-on time Conveyer Belt
       #lfb_TON_ConveyerBelt_Out(IN := NOT "IX_HBW_LightBarrierOutside_I3",
                                 PT := T#300ms);

       // Reload the calibration values - Rack Array
       // A
       "gtyp_HBW".Rack_Pos[1, 1].di_PosRack_Horizontal := "gtyp_HBW".di_PosRack_A1_Horizontal;
       "gtyp_HBW".Rack_Pos[2, 1].di_PosRack_Horizontal := "gtyp_HBW".di_PosRack_A1_Horizontal;
       "gtyp_HBW".Rack_Pos[3, 1].di_PosRack_Horizontal := "gtyp_HBW".di_PosRack_A1_Horizontal;
       // B
       "gtyp_HBW".Rack_Pos[1, 2].di_PosRack_Horizontal := "gtyp_HBW".di_PosRack_B2_Horizontal;
       "gtyp_HBW".Rack_Pos[2, 2].di_PosRack_Horizontal := "gtyp_HBW".di_PosRack_B2_Horizontal;
       "gtyp_HBW".Rack_Pos[3, 2].di_PosRack_Horizontal := "gtyp_HBW".di_PosRack_B2_Horizontal;
       // C
       "gtyp_HBW".Rack_Pos[1, 3].di_PosRack_Horizontal := "gtyp_HBW".di_PosRack_C3_Horizontal;
       "gtyp_HBW".Rack_Pos[2, 3].di_PosRack_Horizontal := "gtyp_HBW".di_PosRack_C3_Horizontal;
       "gtyp_HBW".Rack_Pos[3, 3].di_PosRack_Horizontal := "gtyp_HBW".di_PosRack_C3_Horizontal;
       // 1
       "gtyp_HBW".Rack_Pos[1, 1].di_PosRack_Vertical := "gtyp_HBW".di_PosRack_A1_Vertical;
       "gtyp_HBW".Rack_Pos[1, 2].di_PosRack_Vertical := "gtyp_HBW".di_PosRack_A1_Vertical;
       "gtyp_HBW".Rack_Pos[1, 3].di_PosRack_Vertical := "gtyp_HBW".di_PosRack_A1_Vertical;
       // 2
       "gtyp_HBW".Rack_Pos[2, 1].di_PosRack_Vertical := "gtyp_HBW".di_PosRack_B2_Vertical;
       "gtyp_HBW".Rack_Pos[2, 2].di_PosRack_Vertical := "gtyp_HBW".di_PosRack_B2_Vertical;
       "gtyp_HBW".Rack_Pos[2, 3].di_PosRack_Vertical := "gtyp_HBW".di_PosRack_B2_Vertical;
       // 3
       "gtyp_HBW".Rack_Pos[3, 1].di_PosRack_Vertical := "gtyp_HBW".di_PosRack_C3_Vertical;
       "gtyp_HBW".Rack_Pos[3, 2].di_PosRack_Vertical := "gtyp_HBW".di_PosRack_C3_Vertical;
       "gtyp_HBW".Rack_Pos[3, 3].di_PosRack_Vertical := "gtyp_HBW".di_PosRack_C3_Vertical;

       // step chain HBW
       CASE #li_StepCase OF

           0:  // init
               #lx_Start_TON_Wait := FALSE;
               #lx_Time_Error := FALSE;

               "gtyp_HBW".Horizontal_Axis.x_Start_Positioning := FALSE;
               "gtyp_HBW".Vertical_Axis.x_Start_Positioning := FALSE;
               "gtyp_HBW".Horizontal_Axis.x_Reference := FALSE;
               "gtyp_HBW".Vertical_Axis.x_Reference := FALSE;
               "gtyp_HBW".Horizontal_Axis.i_PWM := -1;
               "gtyp_HBW".Vertical_Axis.i_PWM := -1;

